	W =  -168.557 deg,	P =    -0.849 deg,	R =  -103.190 deg
};
P[1772]{
   GP1:
	UF : 7, UT : 3,	CONFIG : 'F U T, 0, 0, 0',
	X =  -284.464  mm,	Y =   167.284  mm,	Z =     0.271  mm,
	W =  -168.319 deg,	P =    -1.416 deg,	R =  -105.411 deg
};
P[1773]{
   GP1:
	UF : 7, UT : 3,	CONFIG : 'F U T, 0, 0, 0',
	X =  -279.044  mm,	Y =   176.157  mm,	Z =     0.000  mm,
	W =  -167.988 deg,	P =    -1.117 deg,	R =  -107.842 deg
};
P[1774]{
   GP1:
	UF : 7, UT : 3,	CONFIG : 'F U T, 0, 0, 0',
	X =  -279.044  mm,	Y =   176.157  mm,	Z =     0.000  mm,
	W =  -167.988 deg,	P =    -1.117 deg,	R =  -107.842 deg
};
P[1775]{
   GP1:
	UF : 7, UT : 3,	CONFIG : 'F U T, 0, 0, 0',
	X =  -279.044  mm,	Y =   176.157  mm,	Z =     0.000  mm,
	W =  -167.988 deg,	P =    -1.117 deg,	R =  -107.842 deg
};
P[1776]{
   GP1:
	UF : 7, UT : 3,	CONFIG : 'F U T, 0, 0, 0',
	X =  -279.044  mm,	Y =   176.157  mm,	Z =     0.000  mm,
	W =  -167.988 deg,	P =    -1.117 deg,	R =  -107.842 deg
};
P[1777]{
   GP1:
	UF : 7, UT : 3,	CONFIG : 'F U T, 0, 0, 0',
	X =  -233.834  mm,	Y =   232.850  mm,	Z =     0.000  mm,
	W =  -167.362 deg,	P =     0.113 deg,	R =  -119.512 deg
};
P[1778]{
   GP1:
	UF : 7, UT : 3,	CONFIG : 'F U T, 0, 0, 0',
	X =  -233.834  mm,	Y =   232.850  mm,	Z =     0.000  mm,
	W =  -167.362 deg,	P =     0.113 deg,	R =  -119.512 deg
};
P[1779]{
   GP1:
	UF : 7, UT : 3,	CONFIG : 'F U T, 0, 0, 0',
	X =  -233.834  mm,	Y =   232.850  mm,	Z =     0.000  mm,
	W =  -167.362 deg,	P =     0.113 deg,	R =  -119.512 deg
};
P[1780]{
   GP1:
	UF : 7, UT : 3,	CONFIG : 'F U T, 0, 0, 0',
	X =  -233.834  mm,	Y =   232.850  mm,	Z =     0.000  mm,
	W =  -167.362 deg,	P =     0.113 deg,	R =  -119.512 deg
};
P[1781]{
   GP1:
	UF : 7, UT : 3,	CONFIG : 'F U T, 0, 0, 0',
	X =  -223.959  mm,	Y =   242.372  mm,	Z =     0.017  mm,
	W =  -167.363 deg,	P =     0.051 deg,	R =  -122.203 deg
};
P[1782]{
   GP1:
	UF : 7, UT : 3,	CONFIG : 'F U T, 0, 0, 0',
	X =  -213.205  mm,	Y =   251.879  mm,	Z =     0.019  mm,
	W =  -167.357 deg,	P =    -0.013 deg,	R =  -124.752 deg
};
P[1783]{
   GP1:
	UF : 7, UT : 3,	CONFIG : 'F U T, 0, 0, 0',
	X =  -201.087  mm,	Y =   261.652  mm,	Z =     0.013  mm,
	W =  -167.362 deg,	P =    -0.013 deg,	R =  -127.460 deg
};
P[1784]{
   GP1:
	UF : 7, UT : 3,	CONFIG : 'F U T, 0, 0, 0',
	X =  -188.194  mm,	Y =   271.072  mm,	Z =     0.006  mm,
	W =  -167.366 deg,	P =    -0.013 deg,	R =  -130.104 deg
};
P[1785]{
   GP1:
	UF : 7, UT : 3,	CONFIG : 'F U T, 0, 0, 0',
	X =  -174.980  mm,	Y =   279.789  mm,	Z =     0.000  mm,
	W =  -167.371 deg,	P =    -0.013 deg,	R =  -132.787 deg
};
P[1786]{
   GP1:
	UF : 7, UT : 3,	CONFIG : 'F U T, 0, 0, 0',
	X =  -174.980  mm,	Y =   279.789  mm,	Z =     0.000  mm,
	W =  -167.371 deg,	P =    -0.013 deg,	R =  -132.787 deg
};
P[1787]{
   GP1:
	UF : 7, UT : 3,	CONFIG : 'F U T, 0, 0, 0',
	X =  -174.980  mm,	Y =   279.789  mm,	Z =     0.000  mm,
	W =  -167.371 deg,	P =    -0.013 deg,	R =  -132.787 deg
};
P[1788]{
   GP1:
	UF : 7, UT : 3,	CONFIG : 'F U T, 0, 0, 0',
	X =  -174.980  mm,	Y =   279.789  mm,	Z =     0.000  mm,
	W =  -167.371 deg,	P =    -0.013 deg,	R =  -132.787 deg
};
P[1789]{
   GP1:
	UF : 7, UT : 3,	CONFIG : 'F U T, 0, 0, 0',
	X =  -109.648  mm,	Y =   311.249  mm,	Z =     0.000  mm,
	W =  -167.363 deg,	P =     0.003 deg,	R =  -145.199 deg
};
P[1790]{
   GP1:
	UF : 7, UT : 3,	CONFIG : 'F U T, 0, 0, 0',
	X =  -109.648  mm,	Y =   311.249  mm,	Z =     0.000  mm,
	W =  -167.363 deg,	P =     0.003 deg,	R =  -145.199 deg
};
P[1791]{
   GP1:
	UF : 7, UT : 3,	CONFIG : 'F U T, 0, 0, 0',
	X =  -109.648  mm,	Y =   311.249  mm,	Z =     0.000  mm,
	W =  -167.363 deg,	P =     0.003 deg,	R =  -145.199 deg
};
P[1792]{
   GP1:
	UF : 7, UT : 3,	CONFIG : 'F U T, 0, 0, 0',
	X =  -109.648  mm,	Y =   311.249  mm,	Z =     0.000  mm,
	W =  -167.363 deg,	P =     0.003 deg,	R =  -145.199 deg
};
P[1793]{
   GP1:
	UF : 7, UT : 3,	CONFIG : 'F U T, 0, 0, 0',
	X =   -92.942  mm,	Y =   316.644  mm,	Z =     0.000  mm,
	W =  -167.364 deg,	P =     0.002 deg,	R =  -148.612 deg
};
P[1794]{
   GP1:
	UF : 7, UT : 3,	CONFIG : 'F U T, 0, 0, 0',
	X =   -74.994  mm,	Y =   321.366  mm,	Z =     0.000  mm,
	W =  -167.364 deg,	P =     0.001 deg,	R =  -151.812 deg
};
P[1795]{
   GP1:
	UF : 7, UT : 3,	CONFIG : 'F U T, 0, 0, 0',
	X =   -56.916  mm,	Y =   325.063  mm,	Z =     0.000  mm,
	W =  -167.364 deg,	P =     0.001 deg,	R =  -155.040 deg
};
P[1796]{
   GP1:
	UF : 7, UT : 3,	CONFIG : 'F U T, 0, 0, 0',
	X =   -36.254  mm,	Y =   328.016  mm,	Z =     0.000  mm,
	W =  -167.364 deg,	P =     0.000 deg,	R =  -158.080 deg
};
P[1797]{
   GP1:
	UF : 7, UT : 3,	CONFIG : 'F U T, 0, 0, 0',
	X =   -36.254  mm,	Y =   328.016  mm,	Z =     0.000  mm,
	W =  -167.364 deg,	P =     0.000 deg,	R =  -158.080 deg
};
P[1798]{
   GP1:
	UF : 7, UT : 3,	CONFIG : 'F U T, 0, 0, 0',
	X =   -36.254  mm,	Y =   328.016  mm,	Z =     0.000  mm,
	W =  -167.364 deg,	P =     0.000 deg,	R =  -158.080 deg
};
P[1799]{
   GP1:
	UF : 7, UT : 3,	CONFIG : 'F U T, 0, 0, 0',
	X =   -36.254  mm,	Y =   328.016  mm,	Z =     0.000  mm,
	W =  -167.364 deg,	P =     0.000 deg,	R =  -158.080 deg
};
P[1800]{
   GP1:
	UF : 7, UT : 3,	CONFIG : 'F U T, 0, 0, 0',
	X =    36.254  mm,	Y =   328.016  mm,	Z =     0.000  mm,
	W =  -167.363 deg,	P =     0.000 deg,	R =  -171.814 deg
};
P[1801]{
   GP1:
	UF : 7, UT : 3,	CONFIG : 'F U T, 0, 0, 0',
	X =    36.254  mm,	Y =   328.016  mm,	Z =     0.000  mm,
	W =  -167.363 deg,	P =     0.000 deg,	R =  -171.814 deg
};
P[1802]{
   GP1:
	UF : 7, UT : 3,	CONFIG : 'F U T, 0, 0, 0',
	X =    36.254  mm,	Y =   328.016  mm,	Z =     0.000  mm,
	W =  -167.363 deg,	P =     0.000 deg,	R =  -171.814 deg
};
P[1803]{
   GP1:
	UF : 7, UT : 3,	CONFIG : 'F U T, 0, 0, 0',
	X =    36.254  mm,	Y =   328.016  mm,	Z =     0.000  mm,
	W =  -167.363 deg,	P =     0.000 deg,	R =  -171.814 deg
};
P[1804]{
   GP1:
	UF : 7, UT : 3,	CONFIG : 'F U T, 0, 0, 0',
	X =    56.849  mm,	Y =   325.071  mm,	Z =     0.000  mm,
	W =  -167.364 deg,	P =     0.000 deg,	R =  -174.875 deg
};
P[1805]{
   GP1:
	UF : 7, UT : 3,	CONFIG : 'F U T, 0, 0, 0',
	X =    75.000  mm,	Y =   321.364  mm,	Z =     0.000  mm,
	W =  -167.364 deg,	P =     0.000 deg,	R =  -178.084 deg
};
P[1806]{
   GP1:
	UF : 7, UT : 3,	CONFIG : 'F U T, 0, 0, 0',
	X =    92.941  mm,	Y =   316.644  mm,	Z =     0.000  mm,
	W =  -167.364 deg,	P =     0.000 deg,	R =   178.713 deg
};
P[1807]{
   GP1:
	UF : 7, UT : 3,	CONFIG : 'F U T, 0, 0, 0',
	X =   109.648  mm,	Y =   311.249  mm,	Z =     0.000  mm,
	W =  -167.364 deg,	P =     0.000 deg,	R =   175.300 deg
};
P[1808]{
   GP1:
	UF : 7, UT : 3,	CONFIG : 'F U T, 0, 0, 0',
	X =   109.648  mm,	Y =   311.249  mm,	Z =     0.000  mm,
	W =  -167.364 deg,	P =     0.000 deg,	R =   175.300 deg
};
P[1809]{
   GP1:
	UF : 7, UT : 3,	CONFIG : 'F U T, 0, 0, 0',
	X =   109.648  mm,	Y =   311.249  mm,	Z =     0.000  mm,
	W =  -167.364 deg,	P =     0.000 deg,	R =   175.300 deg
};
P[1810]{
   GP1:
	UF : 7, UT : 3,	CONFIG : 'F U T, 0, 0, 0',
	X =   109.648  mm,	Y =   311.249  mm,	Z =     0.000  mm,
	W =  -167.364 deg,	P =     0.000 deg,	R =   175.300 deg
};
P[1811]{
   GP1:
	UF : 7, UT : 3,	CONFIG : 'F U T, 0, 0, 0',
	X =   174.980  mm,	Y =   279.789  mm,	Z =     0.000  mm,
	W =  -167.363 deg,	P =     0.001 deg,	R =   163.044 deg
};
P[1812]{
   GP1:
	UF : 7, UT : 3,	CONFIG : 'F U T, 0, 0, 0',
	X =   174.980  mm,	Y =   279.789  mm,	Z =     0.000  mm,
	W =  -167.363 deg,	P =     0.001 deg,	R =   163.044 deg
};
P[1813]{
   GP1:
	UF : 7, UT : 3,	CONFIG : 'F U T, 0, 0, 0',
	X =   174.980  mm,	Y =   279.789  mm,	Z =     0.000  mm,
	W =  -167.363 deg,	P =     0.001 deg,	R =   163.044 deg
};
P[1814]{
   GP1:
	UF : 7, UT : 3,	CONFIG : 'F U T, 0, 0, 0',
	X =   174.980  mm,	Y =   279.789  mm,	Z =     0.000  mm,
	W =  -167.363 deg,	P =     0.001 deg,	R =   163.044 deg
};
P[1815]{
   GP1:
	UF : 7, UT : 3,	CONFIG : 'F U T, 0, 0, 0',
	X =   190.679  mm,	Y =   269.339  mm,	Z =     0.000  mm,
	W =  -167.364 deg,	P =     0.001 deg,	R =   159.762 deg
};
P[1816]{
   GP1:
	UF : 7, UT : 3,	CONFIG : 'F U T, 0, 0, 0',
	X =   205.753  mm,	Y =   258.007  mm,	Z =     0.000  mm,
	W =  -167.364 deg,	P =     0.000 deg,	R =   156.479 deg
};
P[1817]{
   GP1:
	UF : 7, UT : 3,	CONFIG : 'F U T, 0, 0, 0',
	X =   220.154  mm,	Y =   245.831  mm,	Z =     0.000  mm,
	W =  -167.364 deg,	P =    -0.001 deg,	R =   153.196 deg
};
P[1818]{
   GP1:
	UF : 7, UT : 3,	CONFIG : 'F U T, 0, 0, 0',
	X =   233.834  mm,	Y =   232.850  mm,	Z =     0.000  mm,
	W =  -167.365 deg,	P =    -0.002 deg,	R =   149.914 deg
};
P[1819]{
   GP1:
	UF : 7, UT : 3,	CONFIG : 'F U T, 0, 0, 0',
	X =   233.834  mm,	Y =   232.850  mm,	Z =     0.000  mm,
	W =  -167.365 deg,	P =    -0.002 deg,	R =   149.914 deg
};
P[1820]{
   GP1:
	UF : 7, UT : 3,	CONFIG : 'F U T, 0, 0, 0',
	X =   233.834  mm,	Y =   232.850  mm,	Z =     0.000  mm,
	W =  -167.365 deg,	P =    -0.002 deg,	R =   149.914 deg
};
P[1821]{
   GP1:
	UF : 7, UT : 3,	CONFIG : 'F U T, 0, 0, 0',
	X =   233.834  mm,	Y =   232.850  mm,	Z =     0.000  mm,
	W =  -167.365 deg,	P =    -0.002 deg,	R =   149.914 deg
};
P[1822]{
   GP1:
	UF : 7, UT : 3,	CONFIG : 'F U T, 0, 0, 0',
	X =   279.044  mm,	Y =   176.157  mm,	Z =     0.000  mm,
	W =  -167.363 deg,	P =     0.002 deg,	R =   137.857 deg
};
P[1823]{
   GP1:
	UF : 7, UT : 3,	CONFIG : 'F U T, 0, 0, 0',
	X =   279.044  mm,	Y =   176.157  mm,	Z =     0.000  mm,
	W =  -167.363 deg,	P =     0.002 deg,	R =   137.857 deg
};
P[1824]{
   GP1:
	UF : 7, UT : 3,	CONFIG : 'F U T, 0, 0, 0',
	X =   279.044  mm,	Y =   176.157  mm,	Z =     0.000  mm,
	W =  -167.363 deg,	P =     0.002 deg,	R =   137.857 deg
};
P[1825]{
   GP1:
	UF : 7, UT : 3,	CONFIG : 'F U T, 0, 0, 0',
	X =   279.044  mm,	Y =   176.157  mm,	Z =     0.000  mm,
	W =  -167.363 deg,	P =     0.002 deg,	R =   137.857 deg
};
P[1826]{
   GP1:
	UF : 7, UT : 3,	CONFIG : 'F U T, 0, 0, 0',
	X =   287.893  mm,	Y =   161.305  mm,	Z =     0.000  mm,
	W =  -167.364 deg,	P =     0.001 deg,	R =   134.332 deg
};
P[1827]{
   GP1:
	UF : 7, UT : 3,	CONFIG : 'F U T, 0, 0, 0',
	X =   296.479  mm,	Y =   144.911  mm,	Z =     0.000  mm,
	W =  -167.364 deg,	P =     0.000 deg,	R =   131.099 deg
};
P[1828]{
   GP1:
	UF : 7, UT : 3,	CONFIG : 'F U T, 0, 0, 0',
	X =   304.165  mm,	Y =   128.012  mm,	Z =     0.000  mm,
	W =  -167.364 deg,	P =    -0.001 deg,	R =   127.883 deg
};
P[1829]{
   GP1:
	UF : 7, UT : 3,	CONFIG : 'F U T, 0, 0, 0',
	X =   311.718  mm,	Y =   108.335  mm,	Z =     0.000  mm,
	W =  -167.365 deg,	P =    -0.002 deg,	R =   124.706 deg
};
P[1830]{
   GP1:
	UF : 7, UT : 3,	CONFIG : 'F U T, 0, 0, 0',
	X =   311.718  mm,	Y =   108.335  mm,	Z =     0.000  mm,
	W =  -167.365 deg,	P =    -0.002 deg,	R =   124.706 deg
};
P[1831]{
   GP1:
	UF : 7, UT : 3,	CONFIG : 'F U T, 0, 0, 0',
	X =   311.718  mm,	Y =   108.335  mm,	Z =     0.000  mm,
	W =  -167.365 deg,	P =    -0.002 deg,	R =   124.706 deg
};
P[1832]{
   GP1:
	UF : 7, UT : 3,	CONFIG : 'F U T, 0, 0, 0',
	X =   311.718  mm,	Y =   108.335  mm,	Z =     0.000  mm,
	W =  -167.365 deg,	P =    -0.002 deg,	R =   124.706 deg
};
P[1833]{
   GP1:
	UF : 7, UT : 3,	CONFIG : 'F U T, 0, 0, 0',
	X =   327.850  mm,	Y =    37.642  mm,	Z =     0.000  mm,
	W =  -167.363 deg,	P =     0.001 deg,	R =   111.494 deg
};
P[1834]{
   GP1:
	UF : 7, UT : 3,	CONFIG : 'F U T, 0, 0, 0',
	X =   327.850  mm,	Y =    37.642  mm,	Z =     0.000  mm,
	W =  -167.363 deg,	P =     0.001 deg,	R =   111.494 deg
};
P[1835]{
   GP1:
	UF : 7, UT : 3,	CONFIG : 'F U T, 0, 0, 0',
	X =   327.850  mm,	Y =    37.642  mm,	Z =     0.000  mm,
	W =  -167.363 deg,	P =     0.001 deg,	R =   111.494 deg
};
P[1836]{
   GP1:
	UF : 7, UT : 3,	CONFIG : 'F U T, 0, 0, 0',
	X =   327.850  mm,	Y =    37.642  mm,	Z =     0.000  mm,
	W =  -167.363 deg,	P =     0.001 deg,	R =   111.494 deg
};
P[1837]{
   GP1:
	UF : 7, UT : 3,	CONFIG : 'F U T, 0, 0, 0',
	X =   329.392  mm,	Y =    20.047  mm,	Z =     0.000  mm,
	W =  -167.364 deg,	P =     0.000 deg,	R =   108.496 deg
};
P[1838]{
   GP1:
	UF : 7, UT : 3,	CONFIG : 'F U T, 0, 0, 0',
	X =   330.015  mm,	Y =     0.000  mm,	Z =     0.000  mm,
	W =  -167.364 deg,	P =    -0.001 deg,	R =   105.709 deg
};
P[1839]{
   GP1:
	UF : 7, UT : 3,	CONFIG : 'F U T, 0, 0, 0',
	X =   330.015  mm,	Y =     0.000  mm,	Z =     0.000  mm,
	W =  -167.364 deg,	P =    -0.001 deg,	R =   105.709 deg
};
P[1840]{
   GP1:
	UF : 7, UT : 3,	CONFIG : 'F U T, 0, 0, 0',
	X =   330.015  mm,	Y =     0.000  mm,	Z =     0.000  mm,
	W =  -167.364 deg,	P =    -0.001 deg,	R =   105.709 deg
};
P[1841]{
   GP1:
	UF : 7, UT : 3,	CONFIG : 'F U T, 0, 0, 0',
	X =   330.015  mm,	Y =     0.000  mm,	Z =     0.000  mm,
	W =  -167.364 deg,	P =    -0.001 deg,	R =   105.709 deg
};
P[1842]{
   GP1:
	UF : 7, UT : 3,	CONFIG : 'F U T, 0, 0, 0',
	X =   326.881  mm,	Y =     0.000  mm,	Z =     0.000  mm,
	W =  -167.364 deg,	P =    -0.001 deg,	R =   105.719 deg
};
P[1843]{
   GP1:
	UF : 7, UT : 3,	CONFIG : 'F U T, 0, 0, 0',
	X =   326.881  mm,	Y =     0.000  mm,	Z =     0.000  mm,
	W =  -167.364 deg,	P =    -0.001 deg,	R =   105.719 deg
};
P[1844]{
   GP1:
	UF : 7, UT : 3,	CONFIG : 'F U T, 0, 0, 0',
	X =   326.881  mm,	Y =     0.000  mm,	Z =     0.000  mm,
	W =  -167.364 deg,	P =    -0.001 deg,	R =   105.719 deg
};
P[1845]{
   GP1:
	UF : 7, UT : 3,	CONFIG : 'F U T, 0, 0, 0',
	X =   326.881  mm,	Y =     0.000  mm,	Z =     0.000  mm,
	W =  -167.364 deg,	P =    -0.001 deg,	R =   105.719 deg
};
P[1846]{
   GP1:
	UF : 7, UT : 3,	CONFIG : 'F U T, 0, 0, 0',
	X =   326.322  mm,	Y =    18.789  mm,	Z =     0.000  mm,
	W =  -167.364 deg,	P =     0.000 deg,	R =   108.339 deg
};
P[1847]{
   GP1:
	UF : 7, UT : 3,	CONFIG : 'F U T, 0, 0, 0',
	X =   324.819  mm,	Y =    36.609  mm,	Z =     0.000  mm,
	W =  -167.363 deg,	P =     0.001 deg,	R =   111.080 deg
};
P[1848]{
   GP1:
	UF : 7, UT : 3,	CONFIG : 'F U T, 0, 0, 0',
	X =   324.819  mm,	Y =    36.609  mm,	Z =     0.000  mm,
	W =  -167.363 deg,	P =     0.001 deg,	R =   111.080 deg
};
P[1849]{
   GP1:
	UF : 7, UT : 3,	CONFIG : 'F U T, 0, 0, 0',
	X =   324.819  mm,	Y =    36.609  mm,	Z =     0.000  mm,
	W =  -167.363 deg,	P =     0.001 deg,	R =   111.080 deg
};
P[1850]{
   GP1:
	UF : 7, UT : 3,	CONFIG : 'F U T, 0, 0, 0',
	X =   324.819  mm,	Y =    36.609  mm,	Z =     0.000  mm,
	W =  -167.363 deg,	P =     0.001 deg,	R =   111.080 deg
};
P[1851]{
   GP1:
	UF : 7, UT : 3,	CONFIG : 'F U T, 0, 0, 0',
	X =   308.528  mm,	Y =   107.949  mm,	Z =     0.000  mm,
	W =  -167.365 deg,	P =    -0.002 deg,	R =   124.620 deg
};
P[1852]{
   GP1:
	UF : 7, UT : 3,	CONFIG : 'F U T, 0, 0, 0',
	X =   308.528  mm,	Y =   107.949  mm,	Z =     0.000  mm,
	W =  -167.365 deg,	P =    -0.002 deg,	R =   124.620 deg
};
P[1853]{
   GP1:
	UF : 7, UT : 3,	CONFIG : 'F U T, 0, 0, 0',
	X =   308.528  mm,	Y =   107.949  mm,	Z =     0.000  mm,
	W =  -167.365 deg,	P =    -0.002 deg,	R =   124.620 deg
};
P[1854]{
   GP1:
	UF : 7, UT : 3,	CONFIG : 'F U T, 0, 0, 0',
	X =   308.528  mm,	Y =   107.949  mm,	Z =     0.000  mm,
	W =  -167.365 deg,	P =    -0.002 deg,	R =   124.620 deg
};
P[1855]{
   GP1:
	UF : 7, UT : 3,	CONFIG : 'F U T, 0, 0, 0',
	X =   301.533  mm,	Y =   126.177  mm,	Z =     0.001  mm,
	W =  -167.364 deg,	P =    -0.001 deg,	R =   127.743 deg
};
P[1856]{
   GP1:
	UF : 7, UT : 3,	CONFIG : 'F U T, 0, 0, 0',
	X =   293.998  mm,	Y =   142.847  mm,	Z =     0.000  mm,
	W =  -167.364 deg,	P =     0.000 deg,	R =   130.977 deg
};
P[1857]{
   GP1:
	UF : 7, UT : 3,	CONFIG : 'F U T, 0, 0, 0',
	X =   285.500  mm,	Y =   159.164  mm,	Z =     0.000  mm,
	W =  -167.364 deg,	P =     0.001 deg,	R =   134.192 deg
};
P[1858]{
   GP1:
	UF : 7, UT : 3,	CONFIG : 'F U T, 0, 0, 0',
	X =   276.758  mm,	Y =   173.908  mm,	Z =     0.000  mm,
	W =  -167.363 deg,	P =     0.002 deg,	R =   137.706 deg
};
P[1859]{
   GP1:
	UF : 7, UT : 3,	CONFIG : 'F U T, 0, 0, 0',
	X =   276.758  mm,	Y =   173.908  mm,	Z =     0.000  mm,
	W =  -167.363 deg,	P =     0.002 deg,	R =   137.706 deg
};
P[1860]{
   GP1:
	UF : 7, UT : 3,	CONFIG : 'F U T, 0, 0, 0',
	X =   276.758  mm,	Y =   173.908  mm,	Z =     0.000  mm,
	W =  -167.363 deg,	P =     0.002 deg,	R =   137.706 deg
};
P[1861]{
   GP1:
	UF : 7, UT : 3,	CONFIG : 'F U T, 0, 0, 0',
	X =   276.758  mm,	Y =   173.908  mm,	Z =     0.000  mm,
	W =  -167.363 deg,	P =     0.002 deg,	R =   137.706 deg
};
P[1862]{
   GP1:
	UF : 7, UT : 3,	CONFIG : 'F U T, 0, 0, 0',
	X =   231.131  mm,	Y =   231.120  mm,	Z =     0.000  mm,
	W =  -167.364 deg,	P =    -0.002 deg,	R =   149.652 deg
};
P[1863]{
   GP1:
	UF : 7, UT : 3,	CONFIG : 'F U T, 0, 0, 0',
	X =   231.131  mm,	Y =   231.120  mm,	Z =     0.000  mm,
	W =  -167.364 deg,	P =    -0.002 deg,	R =   149.652 deg
};
P[1864]{
   GP1:
	UF : 7, UT : 3,	CONFIG : 'F U T, 0, 0, 0',
	X =   231.131  mm,	Y =   231.120  mm,	Z =     0.000  mm,
	W =  -167.364 deg,	P =    -0.002 deg,	R =   149.652 deg
};
P[1865]{
   GP1:
	UF : 7, UT : 3,	CONFIG : 'F U T, 0, 0, 0',
	X =   231.131  mm,	Y =   231.120  mm,	Z =     0.000  mm,
	W =  -167.364 deg,	P =    -0.002 deg,	R =   149.652 deg
};
P[1866]{
   GP1:
	UF : 7, UT : 3,	CONFIG : 'F U T, 0, 0, 0',
	X =   218.314  mm,	Y =   243.276  mm,	Z =     0.001  mm,
	W =  -167.364 deg,	P =    -0.001 deg,	R =   153.151 deg
};
P[1867]{
   GP1:
	UF : 7, UT : 3,	CONFIG : 'F U T, 0, 0, 0',
	X =   203.983  mm,	Y =   255.400  mm,	Z =     0.001  mm,
	W =  -167.364 deg,	P =     0.000 deg,	R =   156.409 deg
};
P[1868]{
   GP1:
	UF : 7, UT : 3,	CONFIG : 'F U T, 0, 0, 0',
	X =   189.201  mm,	Y =   266.552  mm,	Z =     0.001  mm,
	W =  -167.364 deg,	P =     0.001 deg,	R =   159.717 deg
};
P[1869]{
   GP1:
	UF : 7, UT : 3,	CONFIG : 'F U T, 0, 0, 0',
	X =   173.895  mm,	Y =   276.767  mm,	Z =     0.000  mm,
	W =  -167.363 deg,	P =     0.002 deg,	R =   163.034 deg
};
P[1870]{
   GP1:
	UF : 7, UT : 3,	CONFIG : 'F U T, 0, 0, 0',
	X =   173.895  mm,	Y =   276.767  mm,	Z =     0.000  mm,
	W =  -167.363 deg,	P =     0.002 deg,	R =   163.034 deg
};
P[1871]{
   GP1:
	UF : 7, UT : 3,	CONFIG : 'F U T, 0, 0, 0',
	X =   173.895  mm,	Y =   276.767  mm,	Z =     0.000  mm,
	W =  -167.363 deg,	P =     0.002 deg,	R =   163.034 deg
};
P[1872]{
   GP1:
	UF : 7, UT : 3,	CONFIG : 'F U T, 0, 0, 0',
	X =   173.895  mm,	Y =   276.767  mm,	Z =     0.000  mm,
	W =  -167.363 deg,	P =     0.002 deg,	R =   163.034 deg
};
P[1873]{
   GP1:
	UF : 7, UT : 3,	CONFIG : 'F U T, 0, 0, 0',
	X =   107.966  mm,	Y =   308.522  mm,	Z =     0.000  mm,
	W =  -167.364 deg,	P =     0.000 deg,	R =   175.671 deg
};
P[1874]{
   GP1:
	UF : 7, UT : 3,	CONFIG : 'F U T, 0, 0, 0',
	X =   107.966  mm,	Y =   308.522  mm,	Z =     0.000  mm,
	W =  -167.364 deg,	P =     0.000 deg,	R =   175.671 deg
};
P[1875]{
   GP1:
	UF : 7, UT : 3,	CONFIG : 'F U T, 0, 0, 0',
	X =   107.966  mm,	Y =   308.522  mm,	Z =     0.000  mm,
	W =  -167.364 deg,	P =     0.000 deg,	R =   175.671 deg
};
P[1876]{
   GP1:
	UF : 7, UT : 3,	CONFIG : 'F U T, 0, 0, 0',
	X =   107.966  mm,	Y =   308.522  mm,	Z =     0.000  mm,
	W =  -167.364 deg,	P =     0.000 deg,	R =   175.671 deg
};
P[1877]{
   GP1:
	UF : 7, UT : 3,	CONFIG : 'F U T, 0, 0, 0',
	X =    91.343  mm,	Y =   313.844  mm,	Z =     0.000  mm,
	W =  -167.364 deg,	P =     0.000 deg,	R =   178.849 deg
};
P[1878]{
   GP1:
	UF : 7, UT : 3,	CONFIG : 'F U T, 0, 0, 0',
	X =    74.067  mm,	Y =   318.365  mm,	Z =     0.000  mm,
	W =  -167.364 deg,	P =     0.000 deg,	R =  -178.042 deg
};
P[1879]{
   GP1:
	UF : 7, UT : 3,	CONFIG : 'F U T, 0, 0, 0',
	X =    56.672  mm,	Y =   321.921  mm,	Z =     0.000  mm,
	W =  -167.364 deg,	P =     0.000 deg,	R =  -174.914 deg
};
P[1880]{
   GP1:
	UF : 7, UT : 3,	CONFIG : 'F U T, 0, 0, 0',
	X =    36.588  mm,	Y =   324.822  mm,	Z =     0.000  mm,
	W =  -167.363 deg,	P =     0.000 deg,	R =  -171.929 deg
};
P[1881]{
   GP1:
	UF : 7, UT : 3,	CONFIG : 'F U T, 0, 0, 0',
	X =    36.588  mm,	Y =   324.822  mm,	Z =     0.000  mm,
	W =  -167.363 deg,	P =     0.000 deg,	R =  -171.929 deg
};
P[1882]{
   GP1:
	UF : 7, UT : 3,	CONFIG : 'F U T, 0, 0, 0',
	X =    36.588  mm,	Y =   324.822  mm,	Z =     0.000  mm,
	W =  -167.363 deg,	P =     0.000 deg,	R =  -171.929 deg
};
P[1883]{
   GP1:
	UF : 7, UT : 3,	CONFIG : 'F U T, 0, 0, 0',
	X =    36.588  mm,	Y =   324.822  mm,	Z =     0.000  mm,
	W =  -167.363 deg,	P =     0.000 deg,	R =  -171.929 deg
};
P[1884]{
   GP1:
	UF : 7, UT : 3,	CONFIG : 'F U T, 0, 0, 0',
	X =   -36.588  mm,	Y =   324.822  mm,	Z =     0.000  mm,
	W =  -167.364 deg,	P =    -0.001 deg,	R =  -157.966 deg
};
P[1885]{
   GP1:
	UF : 7, UT : 3,	CONFIG : 'F U T, 0, 0, 0',
	X =   -36.588  mm,	Y =   324.822  mm,	Z =     0.000  mm,
	W =  -167.364 deg,	P =    -0.001 deg,	R =  -157.966 deg
};
P[1886]{
   GP1:
	UF : 7, UT : 3,	CONFIG : 'F U T, 0, 0, 0',
	X =   -36.588  mm,	Y =   324.822  mm,	Z =     0.000  mm,
	W =  -167.364 deg,	P =    -0.001 deg,	R =  -157.966 deg
};
P[1887]{
   GP1:
	UF : 7, UT : 3,	CONFIG : 'F U T, 0, 0, 0',
	X =   -36.588  mm,	Y =   324.822  mm,	Z =     0.000  mm,
	W =  -167.364 deg,	P =    -0.001 deg,	R =  -157.966 deg
};
P[1888]{
   GP1:
	UF : 7, UT : 3,	CONFIG : 'F U T, 0, 0, 0',
	X =   -56.735  mm,	Y =   321.912  mm,	Z =     0.000  mm,
	W =  -167.364 deg,	P =     0.001 deg,	R =  -154.974 deg
};
P[1889]{
   GP1:
	UF : 7, UT : 3,	CONFIG : 'F U T, 0, 0, 0',
	X =   -74.092  mm,	Y =   318.359  mm,	Z =     0.000  mm,
	W =  -167.364 deg,	P =     0.001 deg,	R =  -151.851 deg
};
P[1890]{
   GP1:
	UF : 7, UT : 3,	CONFIG : 'F U T, 0, 0, 0',
	X =   -91.376  mm,	Y =   313.835  mm,	Z =     0.001  mm,
	W =  -167.363 deg,	P =     0.002 deg,	R =  -148.753 deg
};
P[1891]{
   GP1:
	UF : 7, UT : 3,	CONFIG : 'F U T, 0, 0, 0',
	X =  -107.966  mm,	Y =   308.522  mm,	Z =     0.000  mm,
	W =  -167.363 deg,	P =     0.003 deg,	R =  -145.585 deg
};
P[1892]{
   GP1:
	UF : 7, UT : 3,	CONFIG : 'F U T, 0, 0, 0',
	X =  -107.966  mm,	Y =   308.522  mm,	Z =     0.000  mm,
	W =  -167.363 deg,	P =     0.003 deg,	R =  -145.585 deg
};
P[1893]{
   GP1:
	UF : 7, UT : 3,	CONFIG : 'F U T, 0, 0, 0',
	X =  -107.966  mm,	Y =   308.522  mm,	Z =     0.000  mm,
	W =  -167.363 deg,	P =     0.003 deg,	R =  -145.585 deg
};
P[1894]{
   GP1:
	UF : 7, UT : 3,	CONFIG : 'F U T, 0, 0, 0',
	X =  -107.966  mm,	Y =   308.522  mm,	Z =     0.000  mm,
	W =  -167.363 deg,	P =     0.003 deg,	R =  -145.585 deg
};
P[1895]{
   GP1:
	UF : 7, UT : 3,	CONFIG : 'F U T, 0, 0, 0',
	X =  -173.895  mm,	Y =   276.767  mm,	Z =     0.000  mm,
	W =  -167.370 deg,	P =    -0.015 deg,	R =  -132.924 deg
};
P[1896]{
   GP1:
	UF : 7, UT : 3,	CONFIG : 'F U T, 0, 0, 0',
	X =  -173.895  mm,	Y =   276.767  mm,	Z =     0.000  mm,
	W =  -167.370 deg,	P =    -0.015 deg,	R =  -132.924 deg
};
P[1897]{
   GP1:
	UF : 7, UT : 3,	CONFIG : 'F U T, 0, 0, 0',
	X =  -173.895  mm,	Y =   276.767  mm,	Z =     0.000  mm,
	W =  -167.370 deg,	P =    -0.015 deg,	R =  -132.924 deg
};
P[1898]{
   GP1:
	UF : 7, UT : 3,	CONFIG : 'F U T, 0, 0, 0',
	X =  -173.895  mm,	Y =   276.767  mm,	Z =     0.000  mm,
	W =  -167.370 deg,	P =    -0.015 deg,	R =  -132.924 deg
};
P[1899]{
   GP1:
	UF : 7, UT : 3,	CONFIG : 'F U T, 0, 0, 0',
	X =  -186.182  mm,	Y =   268.655  mm,	Z =     0.005  mm,
	W =  -167.365 deg,	P =    -0.015 deg,	R =  -130.212 deg
};
P[1900]{
   GP1:
	UF : 7, UT : 3,	CONFIG : 'F U T, 0, 0, 0',
	X =  -198.498  mm,	Y =   259.687  mm,	Z =     0.013  mm,
	W =  -167.359 deg,	P =    -0.015 deg,	R =  -127.581 deg
};
P[1901]{
   GP1:
	UF : 7, UT : 3,	CONFIG : 'F U T, 0, 0, 0',
	X =  -210.302  mm,	Y =   250.226  mm,	Z =     0.019  mm,
	W =  -167.354 deg,	P =    -0.016 deg,	R =  -124.938 deg
};
P[1902]{
   GP1:
	UF : 7, UT : 3,	CONFIG : 'F U T, 0, 0, 0',
	X =  -221.274  mm,	Y =   240.579  mm,	Z =     0.017  mm,
	W =  -167.356 deg,	P =     0.051 deg,	R =  -122.320 deg
};
P[1903]{
   GP1:
	UF : 7, UT : 3,	CONFIG : 'F U T, 0, 0, 0',
	X =  -231.131  mm,	Y =   231.120  mm,	Z =     0.000  mm,
	W =  -167.352 deg,	P =     0.114 deg,	R =  -119.469 deg
};
P[1904]{
   GP1:
	UF : 7, UT : 3,	CONFIG : 'F U T, 0, 0, 0',
	X =  -231.131  mm,	Y =   231.120  mm,	Z =     0.000  mm,
	W =  -167.352 deg,	P =     0.114 deg,	R =  -119.469 deg
};
P[1905]{
   GP1:
	UF : 7, UT : 3,	CONFIG : 'F U T, 0, 0, 0',
	X =  -231.131  mm,	Y =   231.120  mm,	Z =     0.000  mm,
	W =  -167.352 deg,	P =     0.114 deg,	R =  -119.469 deg
};
P[1906]{
   GP1:
	UF : 7, UT : 3,	CONFIG : 'F U T, 0, 0, 0',
	X =  -231.131  mm,	Y =   231.120  mm,	Z =     0.000  mm,
	W =  -167.352 deg,	P =     0.114 deg,	R =  -119.469 deg
};
P[1907]{
   GP1:
	UF : 7, UT : 3,	CONFIG : 'F U T, 0, 0, 0',
	X =  -276.758  mm,	Y =   173.908  mm,	Z =     0.000  mm,
	W =  -167.890 deg,	P =    -1.161 deg,	R =  -107.650 deg
};
P[1908]{
   GP1:
	UF : 7, UT : 3,	CONFIG : 'F U T, 0, 0, 0',
	X =  -276.758  mm,	Y =   173.908  mm,	Z =     0.000  mm,
	W =  -167.890 deg,	P =    -1.161 deg,	R =  -107.650 deg
};
P[1909]{
   GP1:
	UF : 7, UT : 3,	CONFIG : 'F U T, 0, 0, 0',
	X =  -276.758  mm,	Y =   173.908  mm,	Z =     0.000  mm,
	W =  -167.890 deg,	P =    -1.161 deg,	R =  -107.650 deg
};
P[1910]{
   GP1:
	UF : 7, UT : 3,	CONFIG : 'F U T, 0, 0, 0',
	X =  -276.758  mm,	Y =   173.908  mm,	Z =     0.000  mm,
	W =  -167.890 deg,	P =    -1.161 deg,	R =  -107.650 deg
};
P[1911]{
   GP1:
	UF : 7, UT : 3,	CONFIG : 'F U T, 0, 0, 0',
	X =  -282.022  mm,	Y =   165.259  mm,	Z =     0.257  mm,
	W =  -168.223 deg,	P =    -1.349 deg,	R =  -105.300 deg
};
P[1912]{
   GP1:
	UF : 7, UT : 3,	CONFIG : 'F U T, 0, 0, 0',
	X =  -288.425  mm,	Y =   153.813  mm,	Z =     0.563  mm,
	W =  -168.481 deg,	P =    -0.762 deg,	R =  -103.051 deg
};
P[1913]{
   GP1:
	UF : 7, UT : 3,	CONFIG : 'F U T, 0, 0, 0',
	X =  -296.971  mm,	Y =   136.562  mm,	Z =     0.670  mm,
	W =  -168.382 deg,	P =     0.631 deg,	R =   -99.690 deg
};
P[1914]{
   GP1:
	UF : 7, UT : 3,	CONFIG : 'F U T, 0, 0, 0',
	X =  -302.664  mm,	Y =   123.431  mm,	Z =     0.424  mm,
	W =  -167.898 deg,	P =     1.805 deg,	R =   -97.151 deg
};
P[1915]{
   GP1:
	UF : 7, UT : 3,	CONFIG : 'F U T, 0, 0, 0',
	X =  -305.358  mm,	Y =   116.596  mm,	Z =     0.206  mm,
	W =  -167.520 deg,	P =     1.756 deg,	R =   -95.843 deg
};
P[1916]{
   GP1:
	UF : 7, UT : 3,	CONFIG : 'F U T, 0, 0, 0',
	X =  -308.528  mm,	Y =   107.949  mm,	Z =     0.000  mm,
	W =  -167.297 deg,	P =     0.804 deg,	R =   -94.511 deg
};
P[1917]{
   GP1:
	UF : 7, UT : 3,	CONFIG : 'F U T, 0, 0, 0',
	X =  -308.528  mm,	Y =   107.949  mm,	Z =     0.000  mm,
	W =  -167.297 deg,	P =     0.804 deg,	R =   -94.511 deg
};
P[1918]{
   GP1:
	UF : 7, UT : 3,	CONFIG : 'F U T, 0, 0, 0',
	X =  -308.528  mm,	Y =   107.949  mm,	Z =     0.000  mm,
	W =  -167.297 deg,	P =     0.804 deg,	R =   -94.511 deg
};
P[1919]{
   GP1:
	UF : 7, UT : 3,	CONFIG : 'F U T, 0, 0, 0',
	X =  -308.528  mm,	Y =   107.949  mm,	Z =     0.000  mm,
	W =  -167.297 deg,	P =     0.804 deg,	R =   -94.511 deg
};
P[1920]{
   GP1:
	UF : 7, UT : 3,	CONFIG : 'F U T, 0, 1, 0',
	X =  -324.819  mm,	Y =    36.609  mm,	Z =     0.000  mm,
	W =  -167.369 deg,	P =    -0.011 deg,	R =   -80.976 deg
};
P[1921]{
   GP1:
	UF : 7, UT : 3,	CONFIG : 'F U T, 0, 1, 0',
	X =  -324.819  mm,	Y =    36.609  mm,	Z =     0.000  mm,
	W =  -167.369 deg,	P =    -0.011 deg,	R =   -80.976 deg
};
P[1922]{
   GP1:
	UF : 7, UT : 3,	CONFIG : 'F U T, 0, 1, 0',
	X =  -324.819  mm,	Y =    36.609  mm,	Z =     0.000  mm,
	W =  -167.369 deg,	P =    -0.011 deg,	R =   -80.976 deg
};
P[1923]{
   GP1:
	UF : 7, UT : 3,	CONFIG : 'F U T, 0, 1, 0',
	X =  -324.819  mm,	Y =    36.609  mm,	Z =     0.000  mm,
	W =  -167.369 deg,	P =    -0.011 deg,	R =   -80.976 deg
};
P[1924]{
   GP1:
	UF : 7, UT : 3,	CONFIG : 'F U T, 0, 1, 0',
	X =  -326.310  mm,	Y =    19.010  mm,	Z =     0.001  mm,
	W =  -167.366 deg,	P =    -0.002 deg,	R =   -78.266 deg
};
P[1925]{
   GP1:
	UF : 7, UT : 3,	CONFIG : 'F U T, 0, 1, 0',
	X =  -326.881  mm,	Y =     0.000  mm,	Z =     0.000  mm,
	W =  -167.362 deg,	P =     0.006 deg,	R =   -75.594 deg
};
P[1926]{
   GP1:
	UF : 7, UT : 3,	CONFIG : 'F U T, 0, 1, 0',
	X =  -326.881  mm,	Y =     0.000  mm,	Z =     0.000  mm,
	W =  -167.362 deg,	P =     0.006 deg,	R =   -75.594 deg
};
P[1927]{
   GP1:
	UF : 7, UT : 3,	CONFIG : 'F U T, 0, 1, 0',
	X =  -326.881  mm,	Y =     0.000  mm,	Z =     0.000  mm,
	W =  -167.362 deg,	P =     0.006 deg,	R =   -75.594 deg
};
P[1928]{
   GP1:
	UF : 7, UT : 3,	CONFIG : 'F U T, 0, 1, 0',
	X =  -326.881  mm,	Y =     0.000  mm,	Z =     0.000  mm,
	W =  -167.362 deg,	P =     0.006 deg,	R =   -75.594 deg
};
P[1929]{
   GP1:
	UF : 7, UT : 3,	CONFIG : 'F U T, 0, 1, 0',
	X =  -323.747  mm,	Y =     0.000  mm,	Z =     0.000  mm,
	W =  -167.362 deg,	P =     0.006 deg,	R =   -75.608 deg
};
P[1930]{
   GP1:
	UF : 7, UT : 3,	CONFIG : 'F U T, 0, 1, 0',
	X =  -323.747  mm,	Y =     0.000  mm,	Z =     0.000  mm,
	W =  -167.362 deg,	P =     0.006 deg,	R =   -75.608 deg
};
P[1931]{
   GP1:
	UF : 7, UT : 3,	CONFIG : 'F U T, 0, 1, 0',
	X =  -323.747  mm,	Y =     0.000  mm,	Z =     0.000  mm,
	W =  -167.362 deg,	P =     0.006 deg,	R =   -75.608 deg
};
P[1932]{
   GP1:
	UF : 7, UT : 3,	CONFIG : 'F U T, 0, 1, 0',
	X =  -323.747  mm,	Y =     0.000  mm,	Z =     0.000  mm,
	W =  -167.362 deg,	P =     0.006 deg,	R =   -75.608 deg
};
P[1933]{
   GP1:
	UF : 7, UT : 3,	CONFIG : 'F U T, 0, 1, 0',
	X =  -323.238  mm,	Y =    17.785  mm,	Z =     0.001  mm,
	W =  -167.365 deg,	P =    -0.002 deg,	R =   -78.103 deg
};
P[1934]{
   GP1:
	UF : 7, UT : 3,	CONFIG : 'F U T, 0, 1, 0',
	X =  -321.754  mm,	Y =    35.852  mm,	Z =     0.000  mm,
	W =  -167.367 deg,	P =    -0.010 deg,	R =   -80.713 deg
};
P[1935]{
   GP1:
	UF : 7, UT : 3,	CONFIG : 'F U T, 0, 1, 0',
	X =  -321.754  mm,	Y =    35.852  mm,	Z =     0.000  mm,
	W =  -167.367 deg,	P =    -0.010 deg,	R =   -80.713 deg
};
P[1936]{
   GP1:
	UF : 7, UT : 3,	CONFIG : 'F U T, 0, 1, 0',
	X =  -321.754  mm,	Y =    35.852  mm,	Z =     0.000  mm,
	W =  -167.367 deg,	P =    -0.010 deg,	R =   -80.713 deg
};
P[1937]{
   GP1:
	UF : 7, UT : 3,	CONFIG : 'F U T, 0, 1, 0',
	X =  -321.754  mm,	Y =    35.852  mm,	Z =     0.000  mm,
	W =  -167.367 deg,	P =    -0.010 deg,	R =   -80.713 deg
};
P[1938]{
   GP1:
	UF : 7, UT : 3,	CONFIG : 'F U T, 0, 0, 0',
	X =  -305.432  mm,	Y =   107.299  mm,	Z =     0.000  mm,
	W =  -167.234 deg,	P =     0.730 deg,	R =   -94.430 deg
};
P[1939]{
   GP1:
	UF : 7, UT : 3,	CONFIG : 'F U T, 0, 0, 0',
	X =  -305.432  mm,	Y =   107.299  mm,	Z =     0.000  mm,
	W =  -167.234 deg,	P =     0.730 deg,	R =   -94.430 deg
};
P[1940]{
   GP1:
	UF : 7, UT : 3,	CONFIG : 'F U T, 0, 0, 0',
	X =  -305.432  mm,	Y =   107.299  mm,	Z =     0.000  mm,
	W =  -167.234 deg,	P =     0.730 deg,	R =   -94.430 deg
};
P[1941]{
   GP1:
	UF : 7, UT : 3,	CONFIG : 'F U T, 0, 0, 0',
	X =  -305.432  mm,	Y =   107.299  mm,	Z =     0.000  mm,
	W =  -167.234 deg,	P =     0.730 deg,	R =   -94.430 deg
};
P[1942]{
   GP1:
	UF : 7, UT : 3,	CONFIG : 'F U T, 0, 0, 0',
	X =  -302.125  mm,	Y =   116.280  mm,	Z =     0.199  mm,
	W =  -167.481 deg,	P =     1.601 deg,	R =   -95.948 deg
};
P[1943]{
   GP1:
	UF : 7, UT : 3,	CONFIG : 'F U T, 0, 0, 0',
	X =  -299.172  mm,	Y =   123.693  mm,	Z =     0.412  mm,
	W =  -167.914 deg,	P =     1.607 deg,	R =   -97.367 deg
};
P[1944]{
   GP1:
	UF : 7, UT : 3,	CONFIG : 'F U T, 0, 0, 0',
	X =  -295.016  mm,	Y =   133.322  mm,	Z =     0.593  mm,
	W =  -168.300 deg,	P =     0.781 deg,	R =   -99.286 deg
};
P[1945]{
   GP1:
	UF : 7, UT : 3,	CONFIG : 'F U T, 0, 0, 0',
	X =  -286.754  mm,	Y =   150.265  mm,	Z =     0.553  mm,
	W =  -168.422 deg,	P =    -0.535 deg,	R =  -102.586 deg
};
P[1946]{
   GP1:
	UF : 7, UT : 3,	CONFIG : 'F U T, 0, 0, 0',
	X =  -279.860  mm,	Y =   162.734  mm,	Z =     0.260  mm,
	W =  -168.144 deg,	P =    -1.256 deg,	R =  -105.066 deg
};
P[1947]{
   GP1:
	UF : 7, UT : 3,	CONFIG : 'F U T, 0, 0, 0',
	X =  -274.323  mm,	Y =   171.896  mm,	Z =     0.000  mm,
	W =  -167.782 deg,	P =    -1.173 deg,	R =  -107.470 deg
};
P[1948]{
   GP1:
	UF : 7, UT : 3,	CONFIG : 'F U T, 0, 0, 0',
	X =  -274.323  mm,	Y =   171.896  mm,	Z =     0.000  mm,
	W =  -167.782 deg,	P =    -1.173 deg,	R =  -107.470 deg
};
P[1949]{
   GP1:
	UF : 7, UT : 3,	CONFIG : 'F U T, 0, 0, 0',
	X =  -274.323  mm,	Y =   171.896  mm,	Z =     0.000  mm,
	W =  -167.782 deg,	P =    -1.173 deg,	R =  -107.470 deg
};
P[1950]{
   GP1:
	UF : 7, UT : 3,	CONFIG : 'F U T, 0, 0, 0',
	X =  -274.323  mm,	Y =   171.896  mm,	Z =     0.000  mm,
	W =  -167.782 deg,	P =    -1.173 deg,	R =  -107.470 deg
};
P[1951]{
   GP1:
	UF : 7, UT : 3,	CONFIG : 'F U T, 0, 0, 0',
	X =  -228.627  mm,	Y =   229.192  mm,	Z =     0.000  mm,
	W =  -167.342 deg,	P =     0.116 deg,	R =  -119.428 deg
};
P[1952]{
   GP1:
	UF : 7, UT : 3,	CONFIG : 'F U T, 0, 0, 0',
	X =  -228.627  mm,	Y =   229.192  mm,	Z =     0.000  mm,
	W =  -167.342 deg,	P =     0.116 deg,	R =  -119.428 deg
};
P[1953]{
   GP1:
	UF : 7, UT : 3,	CONFIG : 'F U T, 0, 0, 0',
	X =  -228.627  mm,	Y =   229.192  mm,	Z =     0.000  mm,
	W =  -167.342 deg,	P =     0.116 deg,	R =  -119.428 deg
};
P[1954]{
   GP1:
	UF : 7, UT : 3,	CONFIG : 'F U T, 0, 0, 0',
	X =  -228.627  mm,	Y =   229.192  mm,	Z =     0.000  mm,
	W =  -167.342 deg,	P =     0.116 deg,	R =  -119.428 deg
};
P[1955]{
   GP1:
	UF : 7, UT : 3,	CONFIG : 'F U T, 0, 0, 0',
	X =  -218.512  mm,	Y =   238.857  mm,	Z =     0.018  mm,
	W =  -167.350 deg,	P =     0.051 deg,	R =  -122.439 deg
};
P[1956]{
   GP1:
	UF : 7, UT : 3,	CONFIG : 'F U T, 0, 0, 0',
	X =  -207.113  mm,	Y =   248.808  mm,	Z =     0.020  mm,
	W =  -167.350 deg,	P =    -0.020 deg,	R =  -125.142 deg
};
P[1957]{
   GP1:
	UF : 7, UT : 3,	CONFIG : 'F U T, 0, 0, 0',
	X =  -189.791  mm,	Y =   262.260  mm,	Z =     0.009  mm,
	W =  -167.360 deg,	P =    -0.017 deg,	R =  -128.976 deg
};
P[1958]{
   GP1:
	UF : 7, UT : 3,	CONFIG : 'F U T, 0, 0, 0',
	X =  -172.572  mm,	Y =   273.895  mm,	Z =     0.000  mm,
	W =  -167.369 deg,	P =    -0.016 deg,	R =  -133.028 deg
};
P[1959]{
   GP1:
	UF : 7, UT : 3,	CONFIG : 'F U T, 0, 0, 0',
	X =  -172.572  mm,	Y =   273.895  mm,	Z =     0.000  mm,
	W =  -167.369 deg,	P =    -0.016 deg,	R =  -133.028 deg
};
P[1960]{
   GP1:
	UF : 7, UT : 3,	CONFIG : 'F U T, 0, 0, 0',
	X =  -172.572  mm,	Y =   273.895  mm,	Z =     0.000  mm,
	W =  -167.369 deg,	P =    -0.016 deg,	R =  -133.028 deg
};
P[1961]{
   GP1:
	UF : 7, UT : 3,	CONFIG : 'F U T, 0, 0, 0',
	X =  -172.572  mm,	Y =   273.895  mm,	Z =     0.000  mm,
	W =  -167.369 deg,	P =    -0.016 deg,	R =  -133.028 deg
};
P[1962]{
   GP1:
	UF : 7, UT : 3,	CONFIG : 'F U T, 0, 0, 0',
	X =  -106.546  mm,	Y =   305.701  mm,	Z =     0.000  mm,
	W =  -167.363 deg,	P =     0.004 deg,	R =  -145.845 deg
};
P[1963]{
   GP1:
	UF : 7, UT : 3,	CONFIG : 'F U T, 0, 0, 0',
	X =  -106.546  mm,	Y =   305.701  mm,	Z =     0.000  mm,
	W =  -167.363 deg,	P =     0.004 deg,	R =  -145.845 deg
};
P[1964]{
   GP1:
	UF : 7, UT : 3,	CONFIG : 'F U T, 0, 0, 0',
	X =  -106.546  mm,	Y =   305.701  mm,	Z =     0.000  mm,
	W =  -167.363 deg,	P =     0.004 deg,	R =  -145.845 deg
};
P[1965]{
   GP1:
	UF : 7, UT : 3,	CONFIG : 'F U T, 0, 0, 0',
	X =  -106.546  mm,	Y =   305.701  mm,	Z =     0.000  mm,
	W =  -167.363 deg,	P =     0.004 deg,	R =  -145.845 deg
};
P[1966]{
   GP1:
	UF : 7, UT : 3,	CONFIG : 'F U T, 0, 0, 0',
	X =   -89.894  mm,	Y =   310.999  mm,	Z =     0.001  mm,
	W =  -167.363 deg,	P =     0.003 deg,	R =  -148.908 deg
};
P[1967]{
   GP1:
	UF : 7, UT : 3,	CONFIG : 'F U T, 0, 0, 0',
	X =   -72.777  mm,	Y =   315.449  mm,	Z =     0.001  mm,
	W =  -167.364 deg,	P =     0.002 deg,	R =  -151.945 deg
};
P[1968]{
   GP1:
	UF : 7, UT : 3,	CONFIG : 'F U T, 0, 0, 0',
	X =   -55.829  mm,	Y =   318.885  mm,	Z =     0.000  mm,
	W =  -167.364 deg,	P =     0.000 deg,	R =  -155.053 deg
};
P[1969]{
   GP1:
	UF : 7, UT : 3,	CONFIG : 'F U T, 0, 0, 0',
	X =   -36.644  mm,	Y =   321.658  mm,	Z =     0.000  mm,
	W =  -167.364 deg,	P =    -0.001 deg,	R =  -157.950 deg
};
P[1970]{
   GP1:
	UF : 7, UT : 3,	CONFIG : 'F U T, 0, 0, 0',
	X =   -36.644  mm,	Y =   321.658  mm,	Z =     0.000  mm,
	W =  -167.364 deg,	P =    -0.001 deg,	R =  -157.950 deg
};
P[1971]{
   GP1:
	UF : 7, UT : 3,	CONFIG : 'F U T, 0, 0, 0',
	X =   -36.644  mm,	Y =   321.658  mm,	Z =     0.000  mm,
	W =  -167.364 deg,	P =    -0.001 deg,	R =  -157.950 deg
};
P[1972]{
   GP1:
	UF : 7, UT : 3,	CONFIG : 'F U T, 0, 0, 0',
	X =   -36.644  mm,	Y =   321.658  mm,	Z =     0.000  mm,
	W =  -167.364 deg,	P =    -0.001 deg,	R =  -157.950 deg
};
P[1973]{
   GP1:
	UF : 7, UT : 3,	CONFIG : 'F U T, 0, 0, 0',
	X =    36.644  mm,	Y =   321.658  mm,	Z =     0.000  mm,
	W =  -167.363 deg,	P =     0.000 deg,	R =  -171.928 deg
};
P[1974]{
   GP1:
	UF : 7, UT : 3,	CONFIG : 'F U T, 0, 0, 0',
	X =    36.644  mm,	Y =   321.658  mm,	Z =     0.000  mm,
	W =  -167.363 deg,	P =     0.000 deg,	R =  -171.928 deg
};
P[1975]{
   GP1:
	UF : 7, UT : 3,	CONFIG : 'F U T, 0, 0, 0',
	X =    36.644  mm,	Y =   321.658  mm,	Z =     0.000  mm,
	W =  -167.363 deg,	P =     0.000 deg,	R =  -171.928 deg
};
P[1976]{
   GP1:
	UF : 7, UT : 3,	CONFIG : 'F U T, 0, 0, 0',
	X =    36.644  mm,	Y =   321.658  mm,	Z =     0.000  mm,
	W =  -167.363 deg,	P =     0.000 deg,	R =  -171.928 deg
};
P[1977]{
   GP1:
	UF : 7, UT : 3,	CONFIG : 'F U T, 0, 0, 0',
	X =    56.062  mm,	Y =   318.845  mm,	Z =     0.000  mm,
	W =  -167.364 deg,	P =     0.000 deg,	R =  -174.895 deg
};
P[1978]{
   GP1:
	UF : 7, UT : 3,	CONFIG : 'F U T, 0, 0, 0',
	X =    73.001  mm,	Y =   315.396  mm,	Z =     0.000  mm,
	W =  -167.364 deg,	P =     0.000 deg,	R =  -177.981 deg
};
P[1979]{
   GP1:
	UF : 7, UT : 3,	CONFIG : 'F U T, 0, 0, 0',
	X =    89.891  mm,	Y =   311.000  mm,	Z =     0.000  mm,
	W =  -167.364 deg,	P =     0.000 deg,	R =   178.977 deg
};
P[1980]{
   GP1:
	UF : 7, UT : 3,	CONFIG : 'F U T, 0, 0, 0',
	X =   106.546  mm,	Y =   305.701  mm,	Z =     0.000  mm,
	W =  -167.364 deg,	P =    -0.001 deg,	R =   175.952 deg
};
P[1981]{
   GP1:
	UF : 7, UT : 3,	CONFIG : 'F U T, 0, 0, 0',
	X =   106.546  mm,	Y =   305.701  mm,	Z =     0.000  mm,
	W =  -167.364 deg,	P =    -0.001 deg,	R =   175.952 deg
};
P[1982]{
   GP1:
	UF : 7, UT : 3,	CONFIG : 'F U T, 0, 0, 0',
	X =   106.546  mm,	Y =   305.701  mm,	Z =     0.000  mm,
	W =  -167.364 deg,	P =    -0.001 deg,	R =   175.952 deg
};
P[1983]{
   GP1:
	UF : 7, UT : 3,	CONFIG : 'F U T, 0, 0, 0',
	X =   106.546  mm,	Y =   305.701  mm,	Z =     0.000  mm,
	W =  -167.364 deg,	P =    -0.001 deg,	R =   175.952 deg
};
P[1984]{
   GP1:
	UF : 7, UT : 3,	CONFIG : 'F U T, 0, 0, 0',
	X =   172.572  mm,	Y =   273.895  mm,	Z =     0.000  mm,
	W =  -167.363 deg,	P =     0.002 deg,	R =   163.224 deg
};
P[1985]{
   GP1:
	UF : 7, UT : 3,	CONFIG : 'F U T, 0, 0, 0',
	X =   172.572  mm,	Y =   273.895  mm,	Z =     0.000  mm,
	W =  -167.363 deg,	P =     0.002 deg,	R =   163.224 deg
};
P[1986]{
   GP1:
	UF : 7, UT : 3,	CONFIG : 'F U T, 0, 0, 0',
	X =   172.572  mm,	Y =   273.895  mm,	Z =     0.000  mm,
	W =  -167.363 deg,	P =     0.002 deg,	R =   163.224 deg
};
P[1987]{
   GP1:
	UF : 7, UT : 3,	CONFIG : 'F U T, 0, 0, 0',
	X =   172.572  mm,	Y =   273.895  mm,	Z =     0.000  mm,
	W =  -167.363 deg,	P =     0.002 deg,	R =   163.224 deg
};
P[1988]{
   GP1:
	UF : 7, UT : 3,	CONFIG : 'F U T, 0, 0, 0',
	X =   187.242  mm,	Y =   264.099  mm,	Z =     0.001  mm,
	W =  -167.364 deg,	P =     0.001 deg,	R =   159.733 deg
};
P[1989]{
   GP1:
	UF : 7, UT : 3,	CONFIG : 'F U T, 0, 0, 0',
	X =   202.010  mm,	Y =   252.966  mm,	Z =     0.001  mm,
	W =  -167.364 deg,	P =     0.000 deg,	R =   156.448 deg
};
P[1990]{
   GP1:
	UF : 7, UT : 3,	CONFIG : 'F U T, 0, 0, 0',
	X =   216.163  mm,	Y =   240.994  mm,	Z =     0.001  mm,
	W =  -167.364 deg,	P =    -0.001 deg,	R =   153.167 deg
};
P[1991]{
   GP1:
	UF : 7, UT : 3,	CONFIG : 'F U T, 0, 0, 0',
	X =   228.627  mm,	Y =   229.192  mm,	Z =     0.000  mm,
	W =  -167.364 deg,	P =    -0.002 deg,	R =   149.541 deg
};
P[1992]{
   GP1:
	UF : 7, UT : 3,	CONFIG : 'F U T, 0, 0, 0',
	X =   228.627  mm,	Y =   229.192  mm,	Z =     0.000  mm,
	W =  -167.364 deg,	P =    -0.002 deg,	R =   149.541 deg
};
P[1993]{
   GP1:
	UF : 7, UT : 3,	CONFIG : 'F U T, 0, 0, 0',
	X =   228.627  mm,	Y =   229.192  mm,	Z =     0.000  mm,
	W =  -167.364 deg,	P =    -0.002 deg,	R =   149.541 deg
};
P[1994]{
   GP1:
	UF : 7, UT : 3,	CONFIG : 'F U T, 0, 0, 0',
	X =   228.627  mm,	Y =   229.192  mm,	Z =     0.000  mm,
	W =  -167.364 deg,	P =    -0.002 deg,	R =   149.541 deg
};
P[1995]{
   GP1:
	UF : 7, UT : 3,	CONFIG : 'F U T, 0, 0, 0',
	X =   274.323  mm,	Y =   171.896  mm,	Z =     0.000  mm,
	W =  -167.363 deg,	P =     0.002 deg,	R =   137.482 deg
};
P[1996]{
   GP1:
	UF : 7, UT : 3,	CONFIG : 'F U T, 0, 0, 0',
	X =   274.323  mm,	Y =   171.896  mm,	Z =     0.000  mm,
	W =  -167.363 deg,	P =     0.002 deg,	R =   137.482 deg
};
P[1997]{
   GP1:
	UF : 7, UT : 3,	CONFIG : 'F U T, 0, 0, 0',
	X =   274.323  mm,	Y =   171.896  mm,	Z =     0.000  mm,
	W =  -167.363 deg,	P =     0.002 deg,	R =   137.482 deg
};
P[1998]{
   GP1:
	UF : 7, UT : 3,	CONFIG : 'F U T, 0, 0, 0',
	X =   274.323  mm,	Y =   171.896  mm,	Z =     0.000  mm,
	W =  -167.363 deg,	P =     0.002 deg,	R =   137.482 deg
};
P[1999]{
   GP1:
	UF : 7, UT : 3,	CONFIG : 'F U T, 0, 0, 0',
	X =   283.027  mm,	Y =   157.162  mm,	Z =     0.000  mm,
	W =  -167.364 deg,	P =     0.001 deg,	R =   134.074 deg
};
P[2000]{
   GP1:
	UF : 7, UT : 3,	CONFIG : 'F U T, 0, 0, 0',
	X =   291.437  mm,	Y =   140.946  mm,	Z =     0.001  mm,
	W =  -167.364 deg,	P =     0.000 deg,	R =   130.910 deg
};
P[2001]{
   GP1:
	UF : 7, UT : 3,	CONFIG : 'F U T, 0, 0, 0',
	X =   298.756  mm,	Y =   124.694  mm,	Z =     0.001  mm,
	W =  -167.364 deg,	P =    -0.001 deg,	R =   127.670 deg
};
P[2002]{
   GP1:
	UF : 7, UT : 3,	CONFIG : 'F U T, 0, 0, 0',
	X =   305.432  mm,	Y =   107.299  mm,	Z =     0.000  mm,
	W =  -167.364 deg,	P =    -0.003 deg,	R =   124.542 deg
};
P[2003]{
   GP1:
	UF : 7, UT : 3,	CONFIG : 'F U T, 0, 0, 0',
	X =   305.432  mm,	Y =   107.299  mm,	Z =     0.000  mm,
	W =  -167.364 deg,	P =    -0.003 deg,	R =   124.542 deg
};
P[2004]{
   GP1:
	UF : 7, UT : 3,	CONFIG : 'F U T, 0, 0, 0',
	X =   305.432  mm,	Y =   107.299  mm,	Z =     0.000  mm,
	W =  -167.364 deg,	P =    -0.003 deg,	R =   124.542 deg
};
P[2005]{
   GP1:
	UF : 7, UT : 3,	CONFIG : 'F U T, 0, 0, 0',
	X =   305.432  mm,	Y =   107.299  mm,	Z =     0.000  mm,
	W =  -167.364 deg,	P =    -0.003 deg,	R =   124.542 deg
};
P[2006]{
   GP1:
	UF : 7, UT : 3,	CONFIG : 'F U T, 0, 0, 0',
	X =   321.754  mm,	Y =    35.852  mm,	Z =     0.000  mm,
	W =  -167.363 deg,	P =     0.001 deg,	R =   110.827 deg
};
P[2007]{
   GP1:
	UF : 7, UT : 3,	CONFIG : 'F U T, 0, 0, 0',
	X =   321.754  mm,	Y =    35.852  mm,	Z =     0.000  mm,
	W =  -167.363 deg,	P =     0.001 deg,	R =   110.827 deg
};
P[2008]{
   GP1:
	UF : 7, UT : 3,	CONFIG : 'F U T, 0, 0, 0',
	X =   321.754  mm,	Y =    35.852  mm,	Z =     0.000  mm,
	W =  -167.363 deg,	P =     0.001 deg,	R =   110.827 deg
};
P[2009]{
   GP1:
	UF : 7, UT : 3,	CONFIG : 'F U T, 0, 0, 0',
	X =   321.754  mm,	Y =    35.852  mm,	Z =     0.000  mm,
	W =  -167.363 deg,	P =     0.001 deg,	R =   110.827 deg
};
P[2010]{
   GP1:
	UF : 7, UT : 3,	CONFIG : 'F U T, 0, 0, 0',
	X =   323.214  mm,	Y =    18.222  mm,	Z =     0.000  mm,
	W =  -167.364 deg,	P =     0.000 deg,	R =   108.254 deg
};
P[2011]{
   GP1:
	UF : 7, UT : 3,	CONFIG : 'F U T, 0, 0, 0',
	X =   323.747  mm,	Y =     0.000  mm,	Z =     0.000  mm,
	W =  -167.364 deg,	P =    -0.001 deg,	R =   105.693 deg
};
P[2012]{
   GP1:
	UF : 7, UT : 3,	CONFIG : 'F U T, 0, 0, 0',
	X =   323.747  mm,	Y =     0.000  mm,	Z =     0.000  mm,
	W =  -167.364 deg,	P =    -0.001 deg,	R =   105.693 deg
};
P[2013]{
   GP1:
	UF : 7, UT : 3,	CONFIG : 'F U T, 0, 0, 0',
	X =   323.747  mm,	Y =     0.000  mm,	Z =     0.000  mm,
	W =  -167.364 deg,	P =    -0.001 deg,	R =   105.693 deg
};
P[2014]{
   GP1:
	UF : 7, UT : 3,	CONFIG : 'F U T, 0, 0, 0',
	X =   323.747  mm,	Y =     0.000  mm,	Z =     0.000  mm,
	W =  -167.364 deg,	P =    -0.001 deg,	R =   105.693 deg
};
P[2015]{
   GP1:
	UF : 7, UT : 3,	CONFIG : 'F U T, 0, 0, 0',
	X =   320.613  mm,	Y =     0.000  mm,	Z =     0.000  mm,
	W =  -167.364 deg,	P =    -0.001 deg,	R =   105.685 deg
};
P[2016]{
   GP1:
	UF : 7, UT : 3,	CONFIG : 'F U T, 0, 0, 0',
	X =   320.613  mm,	Y =     0.000  mm,	Z =     0.000  mm,
	W =  -167.364 deg,	P =    -0.001 deg,	R =   105.685 deg
};
P[2017]{
   GP1:
	UF : 7, UT : 3,	CONFIG : 'F U T, 0, 0, 0',
	X =   320.613  mm,	Y =     0.000  mm,	Z =     0.000  mm,
	W =  -167.364 deg,	P =    -0.001 deg,	R =   105.685 deg
};
P[2018]{
   GP1:
	UF : 7, UT : 3,	CONFIG : 'F U T, 0, 0, 0',
	X =   320.613  mm,	Y =     0.000  mm,	Z =     0.000  mm,
	W =  -167.364 deg,	P =    -0.001 deg,	R =   105.685 deg
};
P[2019]{
   GP1:
	UF : 7, UT : 3,	CONFIG : 'F U T, 0, 0, 0',
	X =   320.087  mm,	Y =    18.011  mm,	Z =     0.000  mm,
	W =  -167.364 deg,	P =     0.000 deg,	R =   108.267 deg
};
P[2020]{
   GP1:
	UF : 7, UT : 3,	CONFIG : 'F U T, 0, 0, 0',
	X =   318.656  mm,	Y =    35.365  mm,	Z =     0.000  mm,
	W =  -167.363 deg,	P =     0.001 deg,	R =   110.739 deg
};
P[2021]{
   GP1:
	UF : 7, UT : 3,	CONFIG : 'F U T, 0, 0, 0',
	X =   318.656  mm,	Y =    35.365  mm,	Z =     0.000  mm,
	W =  -167.363 deg,	P =     0.001 deg,	R =   110.739 deg
};
P[2022]{
   GP1:
	UF : 7, UT : 3,	CONFIG : 'F U T, 0, 0, 0',
	X =   318.656  mm,	Y =    35.365  mm,	Z =     0.000  mm,
	W =  -167.363 deg,	P =     0.001 deg,	R =   110.739 deg
};
P[2023]{
   GP1:
	UF : 7, UT : 3,	CONFIG : 'F U T, 0, 0, 0',
	X =   318.656  mm,	Y =    35.365  mm,	Z =     0.000  mm,
	W =  -167.363 deg,	P =     0.001 deg,	R =   110.739 deg
};
P[2024]{
   GP1:
	UF : 7, UT : 3,	CONFIG : 'F U T, 0, 0, 0',
	X =   302.428  mm,	Y =   106.392  mm,	Z =     0.000  mm,
	W =  -167.364 deg,	P =    -0.003 deg,	R =   124.533 deg
};
P[2025]{
   GP1:
	UF : 7, UT : 3,	CONFIG : 'F U T, 0, 0, 0',
	X =   302.428  mm,	Y =   106.392  mm,	Z =     0.000  mm,
	W =  -167.364 deg,	P =    -0.003 deg,	R =   124.533 deg
};
P[2026]{
   GP1:
	UF : 7, UT : 3,	CONFIG : 'F U T, 0, 0, 0',
	X =   302.428  mm,	Y =   106.392  mm,	Z =     0.000  mm,
	W =  -167.364 deg,	P =    -0.003 deg,	R =   124.533 deg
};
P[2027]{
   GP1:
	UF : 7, UT : 3,	CONFIG : 'F U T, 0, 0, 0',
	X =   302.428  mm,	Y =   106.392  mm,	Z =     0.000  mm,
	W =  -167.364 deg,	P =    -0.003 deg,	R =   124.533 deg
};
P[2028]{
   GP1:
	UF : 7, UT : 3,	CONFIG : 'F U T, 0, 0, 0',
	X =   295.903  mm,	Y =   123.395  mm,	Z =     0.001  mm,
	W =  -167.364 deg,	P =    -0.001 deg,	R =   127.655 deg
};
P[2029]{
   GP1:
	UF : 7, UT : 3,	CONFIG : 'F U T, 0, 0, 0',
	X =   288.703  mm,	Y =   139.400  mm,	Z =     0.001  mm,
	W =  -167.364 deg,	P =     0.000 deg,	R =   130.888 deg
};
P[2030]{
   GP1:
	UF : 7, UT : 3,	CONFIG : 'F U T, 0, 0, 0',
	X =   280.382  mm,	Y =   155.467  mm,	Z =     0.001  mm,
	W =  -167.363 deg,	P =     0.001 deg,	R =   134.031 deg
};
P[2031]{
   GP1:
	UF : 7, UT : 3,	CONFIG : 'F U T, 0, 0, 0',
	X =   271.742  mm,	Y =   170.114  mm,	Z =     0.000  mm,
	W =  -167.363 deg,	P =     0.002 deg,	R =   137.396 deg
};
P[2032]{
   GP1:
	UF : 7, UT : 3,	CONFIG : 'F U T, 0, 0, 0',
	X =   271.742  mm,	Y =   170.114  mm,	Z =     0.000  mm,
	W =  -167.363 deg,	P =     0.002 deg,	R =   137.396 deg
};
P[2033]{
   GP1:
	UF : 7, UT : 3,	CONFIG : 'F U T, 0, 0, 0',
	X =   271.742  mm,	Y =   170.114  mm,	Z =     0.000  mm,
	W =  -167.363 deg,	P =     0.002 deg,	R =   137.396 deg
};
P[2034]{
   GP1:
	UF : 7, UT : 3,	CONFIG : 'F U T, 0, 0, 0',
	X =   271.742  mm,	Y =   170.114  mm,	Z =     0.000  mm,
	W =  -167.363 deg,	P =     0.002 deg,	R =   137.396 deg
};
P[2035]{
   GP1:
	UF : 7, UT : 3,	CONFIG : 'F U T, 0, 0, 0',
	X =   226.314  mm,	Y =   227.073  mm,	Z =     0.000  mm,
	W =  -167.364 deg,	P =    -0.003 deg,	R =   149.494 deg
};
P[2036]{
   GP1:
	UF : 7, UT : 3,	CONFIG : 'F U T, 0, 0, 0',
	X =   226.314  mm,	Y =   227.073  mm,	Z =     0.000  mm,
	W =  -167.364 deg,	P =    -0.003 deg,	R =   149.494 deg
};
P[2037]{
   GP1:
	UF : 7, UT : 3,	CONFIG : 'F U T, 0, 0, 0',
	X =   226.314  mm,	Y =   227.073  mm,	Z =     0.000  mm,
	W =  -167.364 deg,	P =    -0.003 deg,	R =   149.494 deg
};
P[2038]{
   GP1:
	UF : 7, UT : 3,	CONFIG : 'F U T, 0, 0, 0',
	X =   226.314  mm,	Y =   227.073  mm,	Z =     0.000  mm,
	W =  -167.364 deg,	P =    -0.003 deg,	R =   149.494 deg
};
P[2039]{
   GP1:
	UF : 7, UT : 3,	CONFIG : 'F U T, 0, 0, 0',
	X =   214.128  mm,	Y =   238.612  mm,	Z =     0.001  mm,
	W =  -167.364 deg,	P =    -0.002 deg,	R =   153.155 deg
};
P[2040]{
   GP1:
	UF : 7, UT : 3,	CONFIG : 'F U T, 0, 0, 0',
	X =   200.198  mm,	Y =   250.403  mm,	Z =     0.001  mm,
	W =  -167.364 deg,	P =     0.000 deg,	R =   156.441 deg
};
P[2041]{
   GP1:
	UF : 7, UT : 3,	CONFIG : 'F U T, 0, 0, 0',
	X =   185.601  mm,	Y =   261.424  mm,	Z =     0.001  mm,
	W =  -167.363 deg,	P =     0.001 deg,	R =   159.705 deg
};
P[2042]{
   GP1:
	UF : 7, UT : 3,	CONFIG : 'F U T, 0, 0, 0',
	X =   171.020  mm,	Y =   271.169  mm,	Z =     0.000  mm,
	W =  -167.363 deg,	P =     0.002 deg,	R =   163.111 deg
};
P[2043]{
   GP1:
	UF : 7, UT : 3,	CONFIG : 'F U T, 0, 0, 0',
	X =   171.020  mm,	Y =   271.169  mm,	Z =     0.000  mm,
	W =  -167.363 deg,	P =     0.002 deg,	R =   163.111 deg
};
P[2044]{
   GP1:
	UF : 7, UT : 3,	CONFIG : 'F U T, 0, 0, 0',
	X =   171.020  mm,	Y =   271.169  mm,	Z =     0.000  mm,
	W =  -167.363 deg,	P =     0.002 deg,	R =   163.111 deg
};
P[2045]{
   GP1:
	UF : 7, UT : 3,	CONFIG : 'F U T, 0, 0, 0',
	X =   171.020  mm,	Y =   271.169  mm,	Z =     0.000  mm,
	W =  -167.363 deg,	P =     0.002 deg,	R =   163.111 deg
};
P[2046]{
   GP1:
	UF : 7, UT : 3,	CONFIG : 'F U T, 0, 0, 0',
	X =   105.382  mm,	Y =   302.789  mm,	Z =     0.000  mm,
	W =  -167.364 deg,	P =    -0.001 deg,	R =   175.980 deg
};
P[2047]{
   GP1:
	UF : 7, UT : 3,	CONFIG : 'F U T, 0, 0, 0',
	X =   105.382  mm,	Y =   302.789  mm,	Z =     0.000  mm,
	W =  -167.364 deg,	P =    -0.001 deg,	R =   175.980 deg
};
P[2048]{
   GP1:
	UF : 7, UT : 3,	CONFIG : 'F U T, 0, 0, 0',
	X =   105.382  mm,	Y =   302.789  mm,	Z =     0.000  mm,
	W =  -167.364 deg,	P =    -0.001 deg,	R =   175.980 deg
};
P[2049]{
   GP1:
	UF : 7, UT : 3,	CONFIG : 'F U T, 0, 0, 0',
	X =   105.382  mm,	Y =   302.789  mm,	Z =     0.000  mm,
	W =  -167.364 deg,	P =    -0.001 deg,	R =   175.980 deg
};
P[2050]{
   GP1:
	UF : 7, UT : 3,	CONFIG : 'F U T, 0, 0, 0',
	X =    89.059  mm,	Y =   307.979  mm,	Z =     0.000  mm,
	W =  -167.364 deg,	P =     0.000 deg,	R =   179.023 deg
};
P[2051]{
   GP1:
	UF : 7, UT : 3,	CONFIG : 'F U T, 0, 0, 0',
	X =    72.208  mm,	Y =   312.362  mm,	Z =     0.000  mm,
	W =  -167.364 deg,	P =     0.000 deg,	R =  -177.970 deg
};
P[2052]{
   GP1:
	UF : 7, UT : 3,	CONFIG : 'F U T, 0, 0, 0',
	X =    55.598  mm,	Y =   315.746  mm,	Z =     0.000  mm,
	W =  -167.363 deg,	P =     0.000 deg,	R =  -174.901 deg
};
P[2053]{
   GP1:
	UF : 7, UT : 3,	CONFIG : 'F U T, 0, 0, 0',
	X =    36.429  mm,	Y =   318.526  mm,	Z =     0.000  mm,
	W =  -167.363 deg,	P =     0.001 deg,	R =  -171.927 deg
};
P[2054]{
   GP1:
	UF : 7, UT : 3,	CONFIG : 'F U T, 0, 0, 0',
	X =    36.429  mm,	Y =   318.526  mm,	Z =     0.000  mm,
	W =  -167.363 deg,	P =     0.001 deg,	R =  -171.927 deg
};
P[2055]{
   GP1:
	UF : 7, UT : 3,	CONFIG : 'F U T, 0, 0, 0',
	X =    36.429  mm,	Y =   318.526  mm,	Z =     0.000  mm,
	W =  -167.363 deg,	P =     0.001 deg,	R =  -171.927 deg
};
P[2056]{
   GP1:
	UF : 7, UT : 3,	CONFIG : 'F U T, 0, 0, 0',
	X =    36.429  mm,	Y =   318.526  mm,	Z =     0.000  mm,
	W =  -167.363 deg,	P =     0.001 deg,	R =  -171.927 deg
};
P[2057]{
   GP1:
	UF : 7, UT : 3,	CONFIG : 'F U T, 0, 0, 0',
	X =   -36.429  mm,	Y =   318.526  mm,	Z =     0.000  mm,
	W =  -167.364 deg,	P =    -0.001 deg,	R =  -157.992 deg
};
P[2058]{
   GP1:
	UF : 7, UT : 3,	CONFIG : 'F U T, 0, 0, 0',
	X =   -36.429  mm,	Y =   318.526  mm,	Z =     0.000  mm,
	W =  -167.364 deg,	P =    -0.001 deg,	R =  -157.992 deg
};
P[2059]{
   GP1:
	UF : 7, UT : 3,	CONFIG : 'F U T, 0, 0, 0',
	X =   -36.429  mm,	Y =   318.526  mm,	Z =     0.000  mm,
	W =  -167.364 deg,	P =    -0.001 deg,	R =  -157.992 deg
};
P[2060]{
   GP1:
	UF : 7, UT : 3,	CONFIG : 'F U T, 0, 0, 0',
	X =   -36.429  mm,	Y =   318.526  mm,	Z =     0.000  mm,
	W =  -167.364 deg,	P =    -0.001 deg,	R =  -157.992 deg
};
P[2061]{
   GP1:
	UF : 7, UT : 3,	CONFIG : 'F U T, 0, 0, 0',
	X =   -55.427  mm,	Y =   315.774  mm,	Z =     0.000  mm,
	W =  -167.364 deg,	P =     0.000 deg,	R =  -155.025 deg
};
P[2062]{
   GP1:
	UF : 7, UT : 3,	CONFIG : 'F U T, 0, 0, 0',
	X =   -72.033  mm,	Y =   312.407  mm,	Z =     0.001  mm,
	W =  -167.363 deg,	P =     0.002 deg,	R =  -151.941 deg
};
P[2063]{
   GP1:
	UF : 7, UT : 3,	CONFIG : 'F U T, 0, 0, 0',
	X =   -88.851  mm,	Y =   308.037  mm,	Z =     0.001  mm,
	W =  -167.363 deg,	P =     0.003 deg,	R =  -148.939 deg
};
P[2064]{
   GP1:
	UF : 7, UT : 3,	CONFIG : 'F U T, 0, 0, 0',
	X =  -105.382  mm,	Y =   302.789  mm,	Z =     0.000  mm,
	W =  -167.362 deg,	P =     0.004 deg,	R =  -145.933 deg
};
P[2065]{
   GP1:
	UF : 7, UT : 3,	CONFIG : 'F U T, 0, 0, 0',
	X =  -105.382  mm,	Y =   302.789  mm,	Z =     0.000  mm,
	W =  -167.362 deg,	P =     0.004 deg,	R =  -145.933 deg
};
P[2066]{
   GP1:
	UF : 7, UT : 3,	CONFIG : 'F U T, 0, 0, 0',
	X =  -105.382  mm,	Y =   302.789  mm,	Z =     0.000  mm,
	W =  -167.362 deg,	P =     0.004 deg,	R =  -145.933 deg
};
P[2067]{
   GP1:
	UF : 7, UT : 3,	CONFIG : 'F U T, 0, 0, 0',
	X =  -105.382  mm,	Y =   302.789  mm,	Z =     0.000  mm,
	W =  -167.362 deg,	P =     0.004 deg,	R =  -145.933 deg
};
P[2068]{
   GP1:
	UF : 7, UT : 3,	CONFIG : 'F U T, 0, 0, 0',
	X =  -171.020  mm,	Y =   271.169  mm,	Z =     0.000  mm,
	W =  -167.368 deg,	P =    -0.018 deg,	R =  -133.025 deg
};
P[2069]{
   GP1:
	UF : 7, UT : 3,	CONFIG : 'F U T, 0, 0, 0',
	X =  -171.020  mm,	Y =   271.169  mm,	Z =     0.000  mm,
	W =  -167.368 deg,	P =    -0.018 deg,	R =  -133.025 deg
};
P[2070]{
   GP1:
	UF : 7, UT : 3,	CONFIG : 'F U T, 0, 0, 0',
	X =  -171.020  mm,	Y =   271.169  mm,	Z =     0.000  mm,
	W =  -167.368 deg,	P =    -0.018 deg,	R =  -133.025 deg
};
P[2071]{
   GP1:
	UF : 7, UT : 3,	CONFIG : 'F U T, 0, 0, 0',
	X =  -171.020  mm,	Y =   271.169  mm,	Z =     0.000  mm,
	W =  -167.368 deg,	P =    -0.018 deg,	R =  -133.025 deg
};
P[2072]{
   GP1:
	UF : 7, UT : 3,	CONFIG : 'F U T, 0, 0, 0',
	X =  -187.477  mm,	Y =   260.069  mm,	Z =     0.009  mm,
	W =  -167.358 deg,	P =    -0.020 deg,	R =  -129.098 deg
};
P[2073]{
   GP1:
	UF : 7, UT : 3,	CONFIG : 'F U T, 0, 0, 0',
	X =  -204.060  mm,	Y =   247.271  mm,	Z =     0.021  mm,
	W =  -167.348 deg,	P =    -0.023 deg,	R =  -125.372 deg
};
P[2074]{
   GP1:
	UF : 7, UT : 3,	CONFIG : 'F U T, 0, 0, 0',
	X =  -215.835  mm,	Y =   237.057  mm,	Z =     0.019  mm,
	W =  -167.343 deg,	P =     0.050 deg,	R =  -122.549 deg
};
P[2075]{
   GP1:
	UF : 7, UT : 3,	CONFIG : 'F U T, 0, 0, 0',
	X =  -226.314  mm,	Y =   227.073  mm,	Z =     0.000  mm,
	W =  -167.331 deg,	P =     0.117 deg,	R =  -119.398 deg
};
P[2076]{
   GP1:
	UF : 7, UT : 3,	CONFIG : 'F U T, 0, 0, 0',
	X =  -226.314  mm,	Y =   227.073  mm,	Z =     0.000  mm,
	W =  -167.331 deg,	P =     0.117 deg,	R =  -119.398 deg
};
P[2077]{
   GP1:
	UF : 7, UT : 3,	CONFIG : 'F U T, 0, 0, 0',
	X =  -226.314  mm,	Y =   227.073  mm,	Z =     0.000  mm,
	W =  -167.331 deg,	P =     0.117 deg,	R =  -119.398 deg
};
P[2078]{
   GP1:
	UF : 7, UT : 3,	CONFIG : 'F U T, 0, 0, 0',
	X =  -226.314  mm,	Y =   227.073  mm,	Z =     0.000  mm,
	W =  -167.331 deg,	P =     0.117 deg,	R =  -119.398 deg
};
P[2079]{
   GP1:
	UF : 7, UT : 3,	CONFIG : 'F U T, 0, 0, 0',
	X =  -271.742  mm,	Y =   170.114  mm,	Z =     0.000  mm,
	W =  -167.670 deg,	P =    -1.156 deg,	R =  -107.332 deg
};
P[2080]{
   GP1:
	UF : 7, UT : 3,	CONFIG : 'F U T, 0, 0, 0',
	X =  -271.742  mm,	Y =   170.114  mm,	Z =     0.000  mm,
	W =  -167.670 deg,	P =    -1.156 deg,	R =  -107.332 deg
};
P[2081]{
   GP1:
	UF : 7, UT : 3,	CONFIG : 'F U T, 0, 0, 0',
	X =  -271.742  mm,	Y =   170.114  mm,	Z =     0.000  mm,
	W =  -167.670 deg,	P =    -1.156 deg,	R =  -107.332 deg
};
P[2082]{
   GP1:
	UF : 7, UT : 3,	CONFIG : 'F U T, 0, 0, 0',
	X =  -271.742  mm,	Y =   170.114  mm,	Z =     0.000  mm,
	W =  -167.670 deg,	P =    -1.156 deg,	R =  -107.332 deg
};
P[2083]{
   GP1:
	UF : 7, UT : 3,	CONFIG : 'F U T, 0, 0, 0',
	X =  -274.706  mm,	Y =   165.277  mm,	Z =     0.127  mm,
	W =  -167.871 deg,	P =    -1.256 deg,	R =  -106.025 deg
};
P[2084]{
   GP1:
	UF : 7, UT : 3,	CONFIG : 'F U T, 0, 0, 0',
	X =  -281.744  mm,	Y =   152.978  mm,	Z =     0.434  mm,
	W =  -168.275 deg,	P =    -0.791 deg,	R =  -103.504 deg
};
P[2085]{
   GP1:
	UF : 7, UT : 3,	CONFIG : 'F U T, 0, 0, 0',
	X =  -290.413  mm,	Y =   135.821  mm,	Z =     0.560  mm,
	W =  -168.305 deg,	P =     0.505 deg,	R =  -100.002 deg
};
P[2086]{
   GP1:
	UF : 7, UT : 3,	CONFIG : 'F U T, 0, 0, 0',
	X =  -295.433  mm,	Y =   124.518  mm,	Z =     0.411  mm,
	W =  -167.958 deg,	P =     1.369 deg,	R =   -97.800 deg
};
P[2087]{
   GP1:
	UF : 7, UT : 3,	CONFIG : 'F U T, 0, 0, 0',
	X =  -297.236  mm,	Y =   120.134  mm,	Z =     0.303  mm,
	W =  -167.702 deg,	P =     1.518 deg,	R =   -97.034 deg
};
P[2088]{
   GP1:
	UF : 7, UT : 3,	CONFIG : 'F U T, 0, 0, 0',
	X =  -300.508  mm,	Y =   111.723  mm,	Z =     0.091  mm,
	W =  -167.277 deg,	P =     1.178 deg,	R =   -95.358 deg
};
P[2089]{
   GP1:
	UF : 7, UT : 3,	CONFIG : 'F U T, 0, 0, 0',
	X =  -302.428  mm,	Y =   106.392  mm,	Z =     0.000  mm,
	W =  -167.189 deg,	P =     0.643 deg,	R =   -94.404 deg
};
P[2090]{
   GP1:
	UF : 7, UT : 3,	CONFIG : 'F U T, 0, 0, 0',
	X =  -302.428  mm,	Y =   106.392  mm,	Z =     0.000  mm,
	W =  -167.189 deg,	P =     0.643 deg,	R =   -94.404 deg
};
P[2091]{
   GP1:
	UF : 7, UT : 3,	CONFIG : 'F U T, 0, 0, 0',
	X =  -302.428  mm,	Y =   106.392  mm,	Z =     0.000  mm,
	W =  -167.189 deg,	P =     0.643 deg,	R =   -94.404 deg
};
P[2092]{
   GP1:
	UF : 7, UT : 3,	CONFIG : 'F U T, 0, 0, 0',
	X =  -302.428  mm,	Y =   106.392  mm,	Z =     0.000  mm,
	W =  -167.189 deg,	P =     0.643 deg,	R =   -94.404 deg
};
P[2093]{
   GP1:
	UF : 7, UT : 3,	CONFIG : 'F U T, 0, 1, 0',
	X =  -318.656  mm,	Y =    35.365  mm,	Z =     0.000  mm,
	W =  -167.366 deg,	P =    -0.010 deg,	R =   -80.642 deg
};
P[2094]{
   GP1:
	UF : 7, UT : 3,	CONFIG : 'F U T, 0, 1, 0',
	X =  -318.656  mm,	Y =    35.365  mm,	Z =     0.000  mm,
	W =  -167.366 deg,	P =    -0.010 deg,	R =   -80.642 deg
};
P[2095]{
   GP1:
	UF : 7, UT : 3,	CONFIG : 'F U T, 0, 1, 0',
	X =  -318.656  mm,	Y =    35.365  mm,	Z =     0.000  mm,
	W =  -167.366 deg,	P =    -0.010 deg,	R =   -80.642 deg
};
P[2096]{
   GP1:
	UF : 7, UT : 3,	CONFIG : 'F U T, 0, 1, 0',
	X =  -318.656  mm,	Y =    35.365  mm,	Z =     0.000  mm,
	W =  -167.366 deg,	P =    -0.010 deg,	R =   -80.642 deg
};
P[2097]{
   GP1:
	UF : 7, UT : 3,	CONFIG : 'F U T, 0, 1, 0',
	X =  -320.116  mm,	Y =    17.484  mm,	Z =     0.001  mm,
	W =  -167.364 deg,	P =    -0.002 deg,	R =   -78.090 deg
};
P[2098]{
   GP1:
	UF : 7, UT : 3,	CONFIG : 'F U T, 0, 1, 0',
	X =  -320.613  mm,	Y =     0.000  mm,	Z =     0.000  mm,
	W =  -167.362 deg,	P =     0.006 deg,	R =   -75.605 deg
};
P[2099]{
   GP1:
	UF : 7, UT : 3,	CONFIG : 'F U T, 0, 1, 0',
	X =  -320.613  mm,	Y =     0.000  mm,	Z =     0.000  mm,
	W =  -167.362 deg,	P =     0.006 deg,	R =   -75.605 deg
};
P[2100]{
   GP1:
	UF : 7, UT : 3,	CONFIG : 'F U T, 0, 1, 0',
	X =  -320.613  mm,	Y =     0.000  mm,	Z =     0.000  mm,
	W =  -167.362 deg,	P =     0.006 deg,	R =   -75.605 deg
};
P[2101]{
   GP1:
	UF : 7, UT : 3,	CONFIG : 'F U T, 0, 1, 0',
	X =  -320.613  mm,	Y =     0.000  mm,	Z =     0.000  mm,
	W =  -167.362 deg,	P =     0.006 deg,	R =   -75.605 deg
};
P[2102]{
   GP1:
	UF : 7, UT : 3,	CONFIG : 'F U T, 0, 1, 0',
	X =  -317.478  mm,	Y =     0.000  mm,	Z =     0.000  mm,
	W =  -167.362 deg,	P =     0.006 deg,	R =   -75.593 deg
};
P[2103]{
   GP1:
	UF : 7, UT : 3,	CONFIG : 'F U T, 0, 1, 0',
	X =  -317.478  mm,	Y =     0.000  mm,	Z =     0.000  mm,
	W =  -167.362 deg,	P =     0.006 deg,	R =   -75.593 deg
};
P[2104]{
   GP1:
	UF : 7, UT : 3,	CONFIG : 'F U T, 0, 1, 0',
	X =  -317.478  mm,	Y =     0.000  mm,	Z =     0.000  mm,
	W =  -167.362 deg,	P =     0.006 deg,	R =   -75.593 deg
};
P[2105]{
   GP1:
	UF : 7, UT : 3,	CONFIG : 'F U T, 0, 1, 0',
	X =  -317.478  mm,	Y =     0.000  mm,	Z =     0.000  mm,
	W =  -167.362 deg,	P =     0.006 deg,	R =   -75.593 deg
};
P[2106]{
   GP1:
	UF : 7, UT : 3,	CONFIG : 'F U T, 0, 1, 0',
	X =  -316.965  mm,	Y =    17.696  mm,	Z =     0.001  mm,
	W =  -167.364 deg,	P =    -0.002 deg,	R =   -78.136 deg
};
P[2107]{
   GP1:
	UF : 7, UT : 3,	CONFIG : 'F U T, 0, 1, 0',
	X =  -315.526  mm,	Y =    35.143  mm,	Z =     0.000  mm,
	W =  -167.365 deg,	P =    -0.010 deg,	R =   -80.713 deg
};
P[2108]{
   GP1:
	UF : 7, UT : 3,	CONFIG : 'F U T, 0, 1, 0',
	X =  -315.526  mm,	Y =    35.143  mm,	Z =     0.000  mm,
	W =  -167.365 deg,	P =    -0.010 deg,	R =   -80.713 deg
};
P[2109]{
   GP1:
	UF : 7, UT : 3,	CONFIG : 'F U T, 0, 1, 0',
	X =  -315.526  mm,	Y =    35.143  mm,	Z =     0.000  mm,
	W =  -167.365 deg,	P =    -0.010 deg,	R =   -80.713 deg
};
P[2110]{
   GP1:
	UF : 7, UT : 3,	CONFIG : 'F U T, 0, 1, 0',
	X =  -315.526  mm,	Y =    35.143  mm,	Z =     0.000  mm,
	W =  -167.365 deg,	P =    -0.010 deg,	R =   -80.713 deg
};
P[2111]{
   GP1:
	UF : 7, UT : 3,	CONFIG : 'F U T, 0, 0, 0',
	X =  -299.514  mm,	Y =   105.233  mm,	Z =     0.000  mm,
	W =  -167.165 deg,	P =     0.551 deg,	R =   -94.443 deg
};
P[2112]{
   GP1:
	UF : 7, UT : 3,	CONFIG : 'F U T, 0, 0, 0',
	X =  -299.514  mm,	Y =   105.233  mm,	Z =     0.000  mm,
	W =  -167.165 deg,	P =     0.551 deg,	R =   -94.443 deg
};
P[2113]{
   GP1:
	UF : 7, UT : 3,	CONFIG : 'F U T, 0, 0, 0',
	X =  -299.514  mm,	Y =   105.233  mm,	Z =     0.000  mm,
	W =  -167.165 deg,	P =     0.551 deg,	R =   -94.443 deg
};
P[2114]{
   GP1:
	UF : 7, UT : 3,	CONFIG : 'F U T, 0, 0, 0',
	X =  -299.514  mm,	Y =   105.233  mm,	Z =     0.000  mm,
	W =  -167.165 deg,	P =     0.551 deg,	R =   -94.443 deg
};
P[2115]{
   GP1:
	UF : 7, UT : 3,	CONFIG : 'F U T, 0, 0, 0',
	X =  -295.965  mm,	Y =   114.849  mm,	Z =     0.171  mm,
	W =  -167.419 deg,	P =     1.267 deg,	R =   -96.127 deg
};
P[2116]{
   GP1:
	UF : 7, UT : 3,	CONFIG : 'F U T, 0, 0, 0',
	X =  -292.426  mm,	Y =   123.583  mm,	Z =     0.368  mm,
	W =  -167.902 deg,	P =     1.232 deg,	R =   -97.868 deg
};
P[2117]{
   GP1:
	UF : 7, UT : 3,	CONFIG : 'F U T, 0, 0, 0',
	X =  -287.102  mm,	Y =   135.502  mm,	Z =     0.509  mm,
	W =  -168.257 deg,	P =     0.436 deg,	R =  -100.196 deg
};
P[2118]{
   GP1:
	UF : 7, UT : 3,	CONFIG : 'F U T, 0, 0, 0',
	X =  -278.803  mm,	Y =   151.825  mm,	Z =     0.393  mm,
	W =  -168.186 deg,	P =    -0.729 deg,	R =  -103.545 deg
};
P[2119]{
   GP1:
	UF : 7, UT : 3,	CONFIG : 'F U T, 0, 0, 0',
	X =  -271.898  mm,	Y =   163.865  mm,	Z =     0.115  mm,
	W =  -167.761 deg,	P =    -1.183 deg,	R =  -106.031 deg
};
P[2120]{
   GP1:
	UF : 7, UT : 3,	CONFIG : 'F U T, 0, 0, 0',
	X =  -269.018  mm,	Y =   168.557  mm,	Z =     0.000  mm,
	W =  -167.557 deg,	P =    -1.117 deg,	R =  -107.447 deg
};
P[2121]{
   GP1:
	UF : 7, UT : 3,	CONFIG : 'F U T, 0, 0, 0',
	X =  -269.018  mm,	Y =   168.557  mm,	Z =     0.000  mm,
	W =  -167.557 deg,	P =    -1.117 deg,	R =  -107.447 deg
};
P[2122]{
   GP1:
	UF : 7, UT : 3,	CONFIG : 'F U T, 0, 0, 0',
	X =  -269.018  mm,	Y =   168.557  mm,	Z =     0.000  mm,
	W =  -167.557 deg,	P =    -1.117 deg,	R =  -107.447 deg
};
P[2123]{
   GP1:
	UF : 7, UT : 3,	CONFIG : 'F U T, 0, 0, 0',
	X =  -269.018  mm,	Y =   168.557  mm,	Z =     0.000  mm,
	W =  -167.557 deg,	P =    -1.117 deg,	R =  -107.447 deg
};
P[2124]{
   GP1:
	UF : 7, UT : 3,	CONFIG : 'F U T, 0, 0, 0',
	X =  -224.191  mm,	Y =   224.763  mm,	Z =     0.000  mm,
	W =  -167.319 deg,	P =     0.118 deg,	R =  -119.376 deg
};
P[2125]{
   GP1:
	UF : 7, UT : 3,	CONFIG : 'F U T, 0, 0, 0',
	X =  -224.191  mm,	Y =   224.763  mm,	Z =     0.000  mm,
	W =  -167.319 deg,	P =     0.118 deg,	R =  -119.376 deg
};
P[2126]{
   GP1:
	UF : 7, UT : 3,	CONFIG : 'F U T, 0, 0, 0',
	X =  -224.191  mm,	Y =   224.763  mm,	Z =     0.000  mm,
	W =  -167.319 deg,	P =     0.118 deg,	R =  -119.376 deg
};
P[2127]{
   GP1:
	UF : 7, UT : 3,	CONFIG : 'F U T, 0, 0, 0',
	X =  -224.191  mm,	Y =   224.763  mm,	Z =     0.000  mm,
	W =  -167.319 deg,	P =     0.118 deg,	R =  -119.376 deg
};
P[2128]{
   GP1:
	UF : 7, UT : 3,	CONFIG : 'F U T, 0, 0, 0',
	X =  -213.288  mm,	Y =   235.139  mm,	Z =     0.021  mm,
	W =  -167.336 deg,	P =     0.049 deg,	R =  -122.667 deg
};
P[2129]{
   GP1:
	UF : 7, UT : 3,	CONFIG : 'F U T, 0, 0, 0',
	X =  -201.094  mm,	Y =   245.657  mm,	Z =     0.021  mm,
	W =  -167.345 deg,	P =    -0.027 deg,	R =  -125.638 deg
};
P[2130]{
   GP1:
	UF : 7, UT : 3,	CONFIG : 'F U T, 0, 0, 0',
	X =  -185.106  mm,	Y =   257.920  mm,	Z =     0.010  mm,
	W =  -167.356 deg,	P =    -0.023 deg,	R =  -129.232 deg
};
P[2131]{
   GP1:
	UF : 7, UT : 3,	CONFIG : 'F U T, 0, 0, 0',
	X =  -169.241  mm,	Y =   268.585  mm,	Z =     0.000  mm,
	W =  -167.367 deg,	P =    -0.020 deg,	R =  -133.004 deg
};
P[2132]{
   GP1:
	UF : 7, UT : 3,	CONFIG : 'F U T, 0, 0, 0',
	X =  -169.241  mm,	Y =   268.585  mm,	Z =     0.000  mm,
	W =  -167.367 deg,	P =    -0.020 deg,	R =  -133.004 deg
};
P[2133]{
   GP1:
	UF : 7, UT : 3,	CONFIG : 'F U T, 0, 0, 0',
	X =  -169.241  mm,	Y =   268.585  mm,	Z =     0.000  mm,
	W =  -167.367 deg,	P =    -0.020 deg,	R =  -133.004 deg
};
P[2134]{
   GP1:
	UF : 7, UT : 3,	CONFIG : 'F U T, 0, 0, 0',
	X =  -169.241  mm,	Y =   268.585  mm,	Z =     0.000  mm,
	W =  -167.367 deg,	P =    -0.020 deg,	R =  -133.004 deg
};
P[2135]{
   GP1:
	UF : 7, UT : 3,	CONFIG : 'F U T, 0, 0, 0',
	X =  -104.470  mm,	Y =   299.786  mm,	Z =     0.000  mm,
	W =  -167.362 deg,	P =     0.004 deg,	R =  -145.854 deg
};
P[2136]{
   GP1:
	UF : 7, UT : 3,	CONFIG : 'F U T, 0, 0, 0',
	X =  -104.470  mm,	Y =   299.786  mm,	Z =     0.000  mm,
	W =  -167.362 deg,	P =     0.004 deg,	R =  -145.854 deg
};
P[2137]{
   GP1:
	UF : 7, UT : 3,	CONFIG : 'F U T, 0, 0, 0',
	X =  -104.470  mm,	Y =   299.786  mm,	Z =     0.000  mm,
	W =  -167.362 deg,	P =     0.004 deg,	R =  -145.854 deg
};
P[2138]{
   GP1:
	UF : 7, UT : 3,	CONFIG : 'F U T, 0, 0, 0',
	X =  -104.470  mm,	Y =   299.786  mm,	Z =     0.000  mm,
	W =  -167.362 deg,	P =     0.004 deg,	R =  -145.854 deg
};
P[2139]{
   GP1:
	UF : 7, UT : 3,	CONFIG : 'F U T, 0, 0, 0',
	X =   -82.656  mm,	Y =   306.518  mm,	Z =     0.001  mm,
	W =  -167.363 deg,	P =     0.002 deg,	R =  -149.878 deg
};
P[2140]{
   GP1:
	UF : 7, UT : 3,	CONFIG : 'F U T, 0, 0, 0',
	X =   -60.541  mm,	Y =   311.638  mm,	Z =     0.001  mm,
	W =  -167.363 deg,	P =     0.001 deg,	R =  -153.942 deg
};
P[2141]{
   GP1:
	UF : 7, UT : 3,	CONFIG : 'F U T, 0, 0, 0',
	X =   -35.948  mm,	Y =   315.428  mm,	Z =     0.000  mm,
	W =  -167.364 deg,	P =    -0.001 deg,	R =  -157.969 deg
};
P[2142]{
   GP1:
	UF : 7, UT : 3,	CONFIG : 'F U T, 0, 0, 0',
	X =   -35.948  mm,	Y =   315.428  mm,	Z =     0.000  mm,
	W =  -167.364 deg,	P =    -0.001 deg,	R =  -157.969 deg
};
P[2143]{
   GP1:
	UF : 7, UT : 3,	CONFIG : 'F U T, 0, 0, 0',
	X =   -35.948  mm,	Y =   315.428  mm,	Z =     0.000  mm,
	W =  -167.364 deg,	P =    -0.001 deg,	R =  -157.969 deg
};
P[2144]{
   GP1:
	UF : 7, UT : 3,	CONFIG : 'F U T, 0, 0, 0',
	X =   -35.948  mm,	Y =   315.428  mm,	Z =     0.000  mm,
	W =  -167.364 deg,	P =    -0.001 deg,	R =  -157.969 deg
};
P[2145]{
   GP1:
	UF : 7, UT : 3,	CONFIG : 'F U T, 0, 0, 0',
	X =    35.948  mm,	Y =   315.428  mm,	Z =     0.000  mm,
	W =  -167.363 deg,	P =     0.001 deg,	R =  -171.926 deg
};
P[2146]{
   GP1:
	UF : 7, UT : 3,	CONFIG : 'F U T, 0, 0, 0',
	X =    35.948  mm,	Y =   315.428  mm,	Z =     0.000  mm,
	W =  -167.363 deg,	P =     0.001 deg,	R =  -171.926 deg
};
P[2147]{
   GP1:
	UF : 7, UT : 3,	CONFIG : 'F U T, 0, 0, 0',
	X =    35.948  mm,	Y =   315.428  mm,	Z =     0.000  mm,
	W =  -167.363 deg,	P =     0.001 deg,	R =  -171.926 deg
};
P[2148]{
   GP1:
	UF : 7, UT : 3,	CONFIG : 'F U T, 0, 0, 0',
	X =    35.948  mm,	Y =   315.428  mm,	Z =     0.000  mm,
	W =  -167.363 deg,	P =     0.001 deg,	R =  -171.926 deg
};
P[2149]{
   GP1:
	UF : 7, UT : 3,	CONFIG : 'F U T, 0, 0, 0',
	X =    60.517  mm,	Y =   311.643  mm,	Z =     0.000  mm,
	W =  -167.363 deg,	P =     0.000 deg,	R =  -175.940 deg
};
P[2150]{
   GP1:
	UF : 7, UT : 3,	CONFIG : 'F U T, 0, 0, 0',
	X =    82.692  mm,	Y =   306.509  mm,	Z =     0.000  mm,
	W =  -167.364 deg,	P =     0.000 deg,	R =  -179.999 deg
};
P[2151]{
   GP1:
	UF : 7, UT : 3,	CONFIG : 'F U T, 0, 0, 0',
	X =   104.470  mm,	Y =   299.786  mm,	Z =     0.000  mm,
	W =  -167.364 deg,	P =    -0.001 deg,	R =   175.961 deg
};
P[2152]{
   GP1:
	UF : 7, UT : 3,	CONFIG : 'F U T, 0, 0, 0',
	X =   104.470  mm,	Y =   299.786  mm,	Z =     0.000  mm,
	W =  -167.364 deg,	P =    -0.001 deg,	R =   175.961 deg
};
P[2153]{
   GP1:
	UF : 7, UT : 3,	CONFIG : 'F U T, 0, 0, 0',
	X =   104.470  mm,	Y =   299.786  mm,	Z =     0.000  mm,
	W =  -167.364 deg,	P =    -0.001 deg,	R =   175.961 deg
};
P[2154]{
   GP1:
	UF : 7, UT : 3,	CONFIG : 'F U T, 0, 0, 0',
	X =   104.470  mm,	Y =   299.786  mm,	Z =     0.000  mm,
	W =  -167.364 deg,	P =    -0.001 deg,	R =   175.961 deg
};
P[2155]{
   GP1:
	UF : 7, UT : 3,	CONFIG : 'F U T, 0, 0, 0',
	X =   169.241  mm,	Y =   268.585  mm,	Z =     0.000  mm,
	W =  -167.363 deg,	P =     0.002 deg,	R =   163.143 deg
};
P[2156]{
   GP1:
	UF : 7, UT : 3,	CONFIG : 'F U T, 0, 0, 0',
	X =   169.241  mm,	Y =   268.585  mm,	Z =     0.000  mm,
	W =  -167.363 deg,	P =     0.002 deg,	R =   163.143 deg
};
P[2157]{
   GP1:
	UF : 7, UT : 3,	CONFIG : 'F U T, 0, 0, 0',
	X =   169.241  mm,	Y =   268.585  mm,	Z =     0.000  mm,
	W =  -167.363 deg,	P =     0.002 deg,	R =   163.143 deg
};
P[2158]{
   GP1:
	UF : 7, UT : 3,	CONFIG : 'F U T, 0, 0, 0',
	X =   169.241  mm,	Y =   268.585  mm,	Z =     0.000  mm,
	W =  -167.363 deg,	P =     0.002 deg,	R =   163.143 deg
};
P[2159]{
   GP1:
	UF : 7, UT : 3,	CONFIG : 'F U T, 0, 0, 0',
	X =   183.720  mm,	Y =   258.920  mm,	Z =     0.001  mm,
	W =  -167.363 deg,	P =     0.001 deg,	R =   159.718 deg
};
P[2160]{
   GP1:
	UF : 7, UT : 3,	CONFIG : 'F U T, 0, 0, 0',
	X =   198.126  mm,	Y =   248.045  mm,	Z =     0.001  mm,
	W =  -167.364 deg,	P =     0.000 deg,	R =   156.405 deg
};
P[2161]{
   GP1:
	UF : 7, UT : 3,	CONFIG : 'F U T, 0, 0, 0',
	X =   212.090  mm,	Y =   236.233  mm,	Z =     0.001  mm,
	W =  -167.364 deg,	P =    -0.002 deg,	R =   153.153 deg
};
P[2162]{
   GP1:
	UF : 7, UT : 3,	CONFIG : 'F U T, 0, 0, 0',
	X =   224.191  mm,	Y =   224.763  mm,	Z =     0.000  mm,
	W =  -167.364 deg,	P =    -0.003 deg,	R =   149.479 deg
};
P[2163]{
   GP1:
	UF : 7, UT : 3,	CONFIG : 'F U T, 0, 0, 0',
	X =   224.191  mm,	Y =   224.763  mm,	Z =     0.000  mm,
	W =  -167.364 deg,	P =    -0.003 deg,	R =   149.479 deg
};
P[2164]{
   GP1:
	UF : 7, UT : 3,	CONFIG : 'F U T, 0, 0, 0',
	X =   224.191  mm,	Y =   224.763  mm,	Z =     0.000  mm,
	W =  -167.364 deg,	P =    -0.003 deg,	R =   149.479 deg
};
P[2165]{
   GP1:
	UF : 7, UT : 3,	CONFIG : 'F U T, 0, 0, 0',
	X =   224.191  mm,	Y =   224.763  mm,	Z =     0.000  mm,
	W =  -167.364 deg,	P =    -0.003 deg,	R =   149.479 deg
};
P[2166]{
   GP1:
	UF : 7, UT : 3,	CONFIG : 'F U T, 0, 0, 0',
	X =   269.018  mm,	Y =   168.557  mm,	Z =     0.000  mm,
	W =  -167.363 deg,	P =     0.003 deg,	R =   137.473 deg
};
P[2167]{
   GP1:
	UF : 7, UT : 3,	CONFIG : 'F U T, 0, 0, 0',
	X =   269.018  mm,	Y =   168.557  mm,	Z =     0.000  mm,
	W =  -167.363 deg,	P =     0.003 deg,	R =   137.473 deg
};
P[2168]{
   GP1:
	UF : 7, UT : 3,	CONFIG : 'F U T, 0, 0, 0',
	X =   269.018  mm,	Y =   168.557  mm,	Z =     0.000  mm,
	W =  -167.363 deg,	P =     0.003 deg,	R =   137.473 deg
};
P[2169]{
   GP1:
	UF : 7, UT : 3,	CONFIG : 'F U T, 0, 0, 0',
	X =   269.018  mm,	Y =   168.557  mm,	Z =     0.000  mm,
	W =  -167.363 deg,	P =     0.003 deg,	R =   137.473 deg
};
P[2170]{
   GP1:
	UF : 7, UT : 3,	CONFIG : 'F U T, 0, 0, 0',
	X =   277.589  mm,	Y =   154.047  mm,	Z =     0.001  mm,
	W =  -167.363 deg,	P =     0.001 deg,	R =   134.070 deg
};
P[2171]{
   GP1:
	UF : 7, UT : 3,	CONFIG : 'F U T, 0, 0, 0',
	X =   285.805  mm,	Y =   138.195  mm,	Z =     0.001  mm,
	W =  -167.364 deg,	P =     0.000 deg,	R =   130.902 deg
};
P[2172]{
   GP1:
	UF : 7, UT : 3,	CONFIG : 'F U T, 0, 0, 0',
	X =   292.963  mm,	Y =   122.300  mm,	Z =     0.001  mm,
	W =  -167.364 deg,	P =    -0.001 deg,	R =   127.666 deg
};
P[2173]{
   GP1:
	UF : 7, UT : 3,	CONFIG : 'F U T, 0, 0, 0',
	X =   299.514  mm,	Y =   105.233  mm,	Z =     0.000  mm,
	W =  -167.364 deg,	P =    -0.003 deg,	R =   124.545 deg
};
P[2174]{
   GP1:
	UF : 7, UT : 3,	CONFIG : 'F U T, 0, 0, 0',
	X =   299.514  mm,	Y =   105.233  mm,	Z =     0.000  mm,
	W =  -167.364 deg,	P =    -0.003 deg,	R =   124.545 deg
};
P[2175]{
   GP1:
	UF : 7, UT : 3,	CONFIG : 'F U T, 0, 0, 0',
	X =   299.514  mm,	Y =   105.233  mm,	Z =     0.000  mm,
	W =  -167.364 deg,	P =    -0.003 deg,	R =   124.545 deg
};
P[2176]{
   GP1:
	UF : 7, UT : 3,	CONFIG : 'F U T, 0, 0, 0',
	X =   299.514  mm,	Y =   105.233  mm,	Z =     0.000  mm,
	W =  -167.364 deg,	P =    -0.003 deg,	R =   124.545 deg
};
P[2177]{
   GP1:
	UF : 7, UT : 3,	CONFIG : 'F U T, 0, 0, 0',
	X =   315.526  mm,	Y =    35.143  mm,	Z =     0.000  mm,
	W =  -167.363 deg,	P =     0.001 deg,	R =   110.775 deg
};
P[2178]{
   GP1:
	UF : 7, UT : 3,	CONFIG : 'F U T, 0, 0, 0',
	X =   315.526  mm,	Y =    35.143  mm,	Z =     0.000  mm,
	W =  -167.363 deg,	P =     0.001 deg,	R =   110.775 deg
};
P[2179]{
   GP1:
	UF : 7, UT : 3,	CONFIG : 'F U T, 0, 0, 0',
	X =   315.526  mm,	Y =    35.143  mm,	Z =     0.000  mm,
	W =  -167.363 deg,	P =     0.001 deg,	R =   110.775 deg
};
P[2180]{
   GP1:
	UF : 7, UT : 3,	CONFIG : 'F U T, 0, 0, 0',
	X =   315.526  mm,	Y =    35.143  mm,	Z =     0.000  mm,
	W =  -167.363 deg,	P =     0.001 deg,	R =   110.775 deg
};
P[2181]{
   GP1:
	UF : 7, UT : 3,	CONFIG : 'F U T, 0, 0, 0',
	X =   316.958  mm,	Y =    17.828  mm,	Z =     0.000  mm,
	W =  -167.363 deg,	P =     0.000 deg,	R =   108.286 deg
};
P[2182]{
   GP1:
	UF : 7, UT : 3,	CONFIG : 'F U T, 0, 0, 0',
	X =   317.478  mm,	Y =     0.000  mm,	Z =     0.000  mm,
	W =  -167.364 deg,	P =    -0.001 deg,	R =   105.693 deg
};
P[2183]{
   GP1:
	UF : 7, UT : 3,	CONFIG : 'F U T, 0, 0, 0',
	X =   317.478  mm,	Y =     0.000  mm,	Z =     0.000  mm,
	W =  -167.364 deg,	P =    -0.001 deg,	R =   105.693 deg
};
P[2184]{
   GP1:
	UF : 7, UT : 3,	CONFIG : 'F U T, 0, 0, 0',
	X =   317.478  mm,	Y =     0.000  mm,	Z =     0.000  mm,
	W =  -167.364 deg,	P =    -0.001 deg,	R =   105.693 deg
};
P[2185]{
   GP1:
	UF : 7, UT : 3,	CONFIG : 'F U T, 0, 0, 0',
	X =   317.478  mm,	Y =     0.000  mm,	Z =     0.000  mm,
	W =  -167.364 deg,	P =    -0.001 deg,	R =   105.693 deg
};
P[2186]{
   GP1:
	UF : 7, UT : 3,	CONFIG : 'F U T, 0, 0, 0',
	X =   314.344  mm,	Y =     0.000  mm,	Z =     0.000  mm,
	W =  -167.364 deg,	P =    -0.001 deg,	R =   105.705 deg
};
P[2187]{
   GP1:
	UF : 7, UT : 3,	CONFIG : 'F U T, 0, 0, 0',
	X =   314.344  mm,	Y =     0.000  mm,	Z =     0.000  mm,
	W =  -167.364 deg,	P =    -0.001 deg,	R =   105.705 deg
};
P[2188]{
   GP1:
	UF : 7, UT : 3,	CONFIG : 'F U T, 0, 0, 0',
	X =   314.344  mm,	Y =     0.000  mm,	Z =     0.000  mm,
	W =  -167.364 deg,	P =    -0.001 deg,	R =   105.705 deg
};
P[2189]{
   GP1:
	UF : 7, UT : 3,	CONFIG : 'F U T, 0, 0, 0',
	X =   314.344  mm,	Y =     0.000  mm,	Z =     0.000  mm,
	W =  -167.364 deg,	P =    -0.001 deg,	R =   105.705 deg
};
P[2190]{
   GP1:
	UF : 7, UT : 3,	CONFIG : 'F U T, 0, 0, 0',
	X =   313.796  mm,	Y =    18.258  mm,	Z =     0.000  mm,
	W =  -167.363 deg,	P =     0.000 deg,	R =   108.359 deg
};
P[2191]{
   GP1:
	UF : 7, UT : 3,	CONFIG : 'F U T, 0, 0, 0',
	X =   312.363  mm,	Y =    35.193  mm,	Z =     0.000  mm,
	W =  -167.363 deg,	P =     0.001 deg,	R =   111.081 deg
};
P[2192]{
   GP1:
	UF : 7, UT : 3,	CONFIG : 'F U T, 0, 0, 0',
	X =   312.363  mm,	Y =    35.193  mm,	Z =     0.000  mm,
	W =  -167.363 deg,	P =     0.001 deg,	R =   111.081 deg
};
P[2193]{
   GP1:
	UF : 7, UT : 3,	CONFIG : 'F U T, 0, 0, 0',
	X =   312.363  mm,	Y =    35.193  mm,	Z =     0.000  mm,
	W =  -167.363 deg,	P =     0.001 deg,	R =   111.081 deg
};
P[2194]{
   GP1:
	UF : 7, UT : 3,	CONFIG : 'F U T, 0, 0, 0',
	X =   312.363  mm,	Y =    35.193  mm,	Z =     0.000  mm,
	W =  -167.363 deg,	P =     0.001 deg,	R =   111.081 deg
};
P[2195]{
   GP1:
	UF : 7, UT : 3,	CONFIG : 'F U T, 0, 0, 0',
	X =   296.692  mm,	Y =   103.818  mm,	Z =     0.000  mm,
	W =  -167.364 deg,	P =    -0.003 deg,	R =   124.612 deg
};
P[2196]{
   GP1:
	UF : 7, UT : 3,	CONFIG : 'F U T, 0, 0, 0',
	X =   296.692  mm,	Y =   103.818  mm,	Z =     0.000  mm,
	W =  -167.364 deg,	P =    -0.003 deg,	R =   124.612 deg
};
P[2197]{
   GP1:
	UF : 7, UT : 3,	CONFIG : 'F U T, 0, 0, 0',
	X =   296.692  mm,	Y =   103.818  mm,	Z =     0.000  mm,
	W =  -167.364 deg,	P =    -0.003 deg,	R =   124.612 deg
};
P[2198]{
   GP1:
	UF : 7, UT : 3,	CONFIG : 'F U T, 0, 0, 0',
	X =   296.692  mm,	Y =   103.818  mm,	Z =     0.000  mm,
	W =  -167.364 deg,	P =    -0.003 deg,	R =   124.612 deg
};
P[2199]{
   GP1:
	UF : 7, UT : 3,	CONFIG : 'F U T, 0, 0, 0',
	X =   289.976  mm,	Y =   121.319  mm,	Z =     0.001  mm,
	W =  -167.364 deg,	P =    -0.001 deg,	R =   127.739 deg
};
P[2200]{
   GP1:
	UF : 7, UT : 3,	CONFIG : 'F U T, 0, 0, 0',
	X =   282.724  mm,	Y =   137.365  mm,	Z =     0.001  mm,
	W =  -167.363 deg,	P =     0.000 deg,	R =   130.985 deg
};
P[2201]{
   GP1:
	UF : 7, UT : 3,	CONFIG : 'F U T, 0, 0, 0',
	X =   274.534  mm,	Y =   153.088  mm,	Z =     0.001  mm,
	W =  -167.363 deg,	P =     0.001 deg,	R =   134.198 deg
};
P[2202]{
   GP1:
	UF : 7, UT : 3,	CONFIG : 'F U T, 0, 0, 0',
	X =   266.148  mm,	Y =   167.232  mm,	Z =     0.000  mm,
	W =  -167.362 deg,	P =     0.003 deg,	R =   137.749 deg
};
P[2203]{
   GP1:
	UF : 7, UT : 3,	CONFIG : 'F U T, 0, 0, 0',
	X =   266.148  mm,	Y =   167.232  mm,	Z =     0.000  mm,
	W =  -167.362 deg,	P =     0.003 deg,	R =   137.749 deg
};
P[2204]{
   GP1:
	UF : 7, UT : 3,	CONFIG : 'F U T, 0, 0, 0',
	X =   266.148  mm,	Y =   167.232  mm,	Z =     0.000  mm,
	W =  -167.362 deg,	P =     0.003 deg,	R =   137.749 deg
};
P[2205]{
   GP1:
	UF : 7, UT : 3,	CONFIG : 'F U T, 0, 0, 0',
	X =   266.148  mm,	Y =   167.232  mm,	Z =     0.000  mm,
	W =  -167.362 deg,	P =     0.003 deg,	R =   137.749 deg
};
P[2206]{
   GP1:
	UF : 7, UT : 3,	CONFIG : 'F U T, 0, 0, 0',
	X =   222.261  mm,	Y =   222.261  mm,	Z =     0.000  mm,
	W =  -167.364 deg,	P =    -0.003 deg,	R =   149.599 deg
};
P[2207]{
   GP1:
	UF : 7, UT : 3,	CONFIG : 'F U T, 0, 0, 0',
	X =   222.261  mm,	Y =   222.261  mm,	Z =     0.000  mm,
	W =  -167.364 deg,	P =    -0.003 deg,	R =   149.599 deg
};
P[2208]{
   GP1:
	UF : 7, UT : 3,	CONFIG : 'F U T, 0, 0, 0',
	X =   222.261  mm,	Y =   222.261  mm,	Z =     0.000  mm,
	W =  -167.364 deg,	P =    -0.003 deg,	R =   149.599 deg
};
P[2209]{
   GP1:
	UF : 7, UT : 3,	CONFIG : 'F U T, 0, 0, 0',
	X =   222.261  mm,	Y =   222.261  mm,	Z =     0.000  mm,
	W =  -167.364 deg,	P =    -0.003 deg,	R =   149.599 deg
};
P[2210]{
   GP1:
	UF : 7, UT : 3,	CONFIG : 'F U T, 0, 0, 0',
	X =   209.897  mm,	Y =   233.994  mm,	Z =     0.001  mm,
	W =  -167.364 deg,	P =    -0.002 deg,	R =   153.153 deg
};
P[2211]{
   GP1:
	UF : 7, UT : 3,	CONFIG : 'F U T, 0, 0, 0',
	X =   195.899  mm,	Y =   245.814  mm,	Z =     0.001  mm,
	W =  -167.363 deg,	P =     0.000 deg,	R =   156.411 deg
};
P[2212]{
   GP1:
	UF : 7, UT : 3,	CONFIG : 'F U T, 0, 0, 0',
	X =   181.688  mm,	Y =   256.510  mm,	Z =     0.001  mm,
	W =  -167.363 deg,	P =     0.001 deg,	R =   159.771 deg
};
P[2213]{
   GP1:
	UF : 7, UT : 3,	CONFIG : 'F U T, 0, 0, 0',
	X =   167.232  mm,	Y =   266.148  mm,	Z =     0.000  mm,
	W =  -167.362 deg,	P =     0.002 deg,	R =   163.242 deg
};
P[2214]{
   GP1:
	UF : 7, UT : 3,	CONFIG : 'F U T, 0, 0, 0',
	X =   167.232  mm,	Y =   266.148  mm,	Z =     0.000  mm,
	W =  -167.362 deg,	P =     0.002 deg,	R =   163.242 deg
};
P[2215]{
   GP1:
	UF : 7, UT : 3,	CONFIG : 'F U T, 0, 0, 0',
	X =   167.232  mm,	Y =   266.148  mm,	Z =     0.000  mm,
	W =  -167.362 deg,	P =     0.002 deg,	R =   163.242 deg
};
P[2216]{
   GP1:
	UF : 7, UT : 3,	CONFIG : 'F U T, 0, 0, 0',
	X =   167.232  mm,	Y =   266.148  mm,	Z =     0.000  mm,
	W =  -167.362 deg,	P =     0.002 deg,	R =   163.242 deg
};
P[2217]{
   GP1:
	UF : 7, UT : 3,	CONFIG : 'F U T, 0, 0, 0',
	X =   103.816  mm,	Y =   296.692  mm,	Z =     0.000  mm,
	W =  -167.364 deg,	P =    -0.001 deg,	R =   175.609 deg
};
P[2218]{
   GP1:
	UF : 7, UT : 3,	CONFIG : 'F U T, 0, 0, 0',
	X =   103.816  mm,	Y =   296.692  mm,	Z =     0.000  mm,
	W =  -167.364 deg,	P =    -0.001 deg,	R =   175.609 deg
};
P[2219]{
   GP1:
	UF : 7, UT : 3,	CONFIG : 'F U T, 0, 0, 0',
	X =   103.816  mm,	Y =   296.692  mm,	Z =     0.000  mm,
	W =  -167.364 deg,	P =    -0.001 deg,	R =   175.609 deg
};
P[2220]{
   GP1:
	UF : 7, UT : 3,	CONFIG : 'F U T, 0, 0, 0',
	X =   103.816  mm,	Y =   296.692  mm,	Z =     0.000  mm,
	W =  -167.364 deg,	P =    -0.001 deg,	R =   175.609 deg
};
P[2221]{
   GP1:
	UF : 7, UT : 3,	CONFIG : 'F U T, 0, 0, 0',
	X =    87.953  mm,	Y =   301.775  mm,	Z =     0.000  mm,
	W =  -167.364 deg,	P =    -0.001 deg,	R =   178.852 deg
};
P[2222]{
   GP1:
	UF : 7, UT : 3,	CONFIG : 'F U T, 0, 0, 0',
	X =    71.164  mm,	Y =   306.169  mm,	Z =     0.000  mm,
	W =  -167.363 deg,	P =     0.000 deg,	R =  -178.042 deg
};
P[2223]{
   GP1:
	UF : 7, UT : 3,	CONFIG : 'F U T, 0, 0, 0',
	X =    54.389  mm,	Y =   309.594  mm,	Z =     0.000  mm,
	W =  -167.363 deg,	P =     0.000 deg,	R =  -174.890 deg
};
P[2224]{
   GP1:
	UF : 7, UT : 3,	CONFIG : 'F U T, 0, 0, 0',
	X =    35.197  mm,	Y =   312.362  mm,	Z =     0.000  mm,
	W =  -167.363 deg,	P =     0.001 deg,	R =  -171.894 deg
};
P[2225]{
   GP1:
	UF : 7, UT : 3,	CONFIG : 'F U T, 0, 0, 0',
	X =    35.197  mm,	Y =   312.362  mm,	Z =     0.000  mm,
	W =  -167.363 deg,	P =     0.001 deg,	R =  -171.894 deg
};
P[2226]{
   GP1:
	UF : 7, UT : 3,	CONFIG : 'F U T, 0, 0, 0',
	X =    35.197  mm,	Y =   312.362  mm,	Z =     0.000  mm,
	W =  -167.363 deg,	P =     0.001 deg,	R =  -171.894 deg
};
P[2227]{
   GP1:
	UF : 7, UT : 3,	CONFIG : 'F U T, 0, 0, 0',
	X =    35.197  mm,	Y =   312.362  mm,	Z =     0.000  mm,
	W =  -167.363 deg,	P =     0.001 deg,	R =  -171.894 deg
};
P[2228]{
   GP1:
	UF : 7, UT : 3,	CONFIG : 'F U T, 0, 0, 0',
	X =   -35.197  mm,	Y =   312.362  mm,	Z =     0.000  mm,
	W =  -167.364 deg,	P =    -0.001 deg,	R =  -157.993 deg
};
P[2229]{
   GP1:
	UF : 7, UT : 3,	CONFIG : 'F U T, 0, 0, 0',
	X =   -35.197  mm,	Y =   312.362  mm,	Z =     0.000  mm,
	W =  -167.364 deg,	P =    -0.001 deg,	R =  -157.993 deg
};
P[2230]{
   GP1:
	UF : 7, UT : 3,	CONFIG : 'F U T, 0, 0, 0',
	X =   -35.197  mm,	Y =   312.362  mm,	Z =     0.000  mm,
	W =  -167.364 deg,	P =    -0.001 deg,	R =  -157.993 deg
};
P[2231]{
   GP1:
	UF : 7, UT : 3,	CONFIG : 'F U T, 0, 0, 0',
	X =   -35.197  mm,	Y =   312.362  mm,	Z =     0.000  mm,
	W =  -167.364 deg,	P =    -0.001 deg,	R =  -157.993 deg
};
P[2232]{
   GP1:
	UF : 7, UT : 3,	CONFIG : 'F U T, 0, 0, 0',
	X =   -54.397  mm,	Y =   309.592  mm,	Z =     0.001  mm,
	W =  -167.363 deg,	P =     0.000 deg,	R =  -154.999 deg
};
P[2233]{
   GP1:
	UF : 7, UT : 3,	CONFIG : 'F U T, 0, 0, 0',
	X =   -71.123  mm,	Y =   306.179  mm,	Z =     0.001  mm,
	W =  -167.363 deg,	P =     0.002 deg,	R =  -151.872 deg
};
P[2234]{
   GP1:
	UF : 7, UT : 3,	CONFIG : 'F U T, 0, 0, 0',
	X =   -87.830  mm,	Y =   301.810  mm,	Z =     0.001  mm,
	W =  -167.362 deg,	P =     0.003 deg,	R =  -148.771 deg
};
P[2235]{
   GP1:
	UF : 7, UT : 3,	CONFIG : 'F U T, 0, 0, 0',
	X =  -103.816  mm,	Y =   296.692  mm,	Z =     0.000  mm,
	W =  -167.361 deg,	P =     0.004 deg,	R =  -145.598 deg
};
P[2236]{
   GP1:
	UF : 7, UT : 3,	CONFIG : 'F U T, 0, 0, 0',
	X =  -103.816  mm,	Y =   296.692  mm,	Z =     0.000  mm,
	W =  -167.361 deg,	P =     0.004 deg,	R =  -145.598 deg
};
P[2237]{
   GP1:
	UF : 7, UT : 3,	CONFIG : 'F U T, 0, 0, 0',
	X =  -103.816  mm,	Y =   296.692  mm,	Z =     0.000  mm,
	W =  -167.361 deg,	P =     0.004 deg,	R =  -145.598 deg
};
P[2238]{
   GP1:
	UF : 7, UT : 3,	CONFIG : 'F U T, 0, 0, 0',
	X =  -103.816  mm,	Y =   296.692  mm,	Z =     0.000  mm,
	W =  -167.361 deg,	P =     0.004 deg,	R =  -145.598 deg
};
P[2239]{
   GP1:
	UF : 7, UT : 3,	CONFIG : 'F U T, 0, 0, 0',
	X =  -167.232  mm,	Y =   266.148  mm,	Z =     0.000  mm,
	W =  -167.365 deg,	P =    -0.022 deg,	R =  -132.938 deg
};
P[2240]{
   GP1:
	UF : 7, UT : 3,	CONFIG : 'F U T, 0, 0, 0',
	X =  -167.232  mm,	Y =   266.148  mm,	Z =     0.000  mm,
	W =  -167.365 deg,	P =    -0.022 deg,	R =  -132.938 deg
};
P[2241]{
   GP1:
	UF : 7, UT : 3,	CONFIG : 'F U T, 0, 0, 0',
	X =  -167.232  mm,	Y =   266.148  mm,	Z =     0.000  mm,
	W =  -167.365 deg,	P =    -0.022 deg,	R =  -132.938 deg
};
P[2242]{
   GP1:
	UF : 7, UT : 3,	CONFIG : 'F U T, 0, 0, 0',
	X =  -167.232  mm,	Y =   266.148  mm,	Z =     0.000  mm,
	W =  -167.365 deg,	P =    -0.022 deg,	R =  -132.938 deg
};
P[2243]{
   GP1:
	UF : 7, UT : 3,	CONFIG : 'F U T, 0, 0, 0',
	X =  -183.114  mm,	Y =   255.488  mm,	Z =     0.011  mm,
	W =  -167.354 deg,	P =    -0.024 deg,	R =  -129.291 deg
};
P[2244]{
   GP1:
	UF : 7, UT : 3,	CONFIG : 'F U T, 0, 0, 0',
	X =  -198.763  mm,	Y =   243.515  mm,	Z =     0.023  mm,
	W =  -167.343 deg,	P =    -0.029 deg,	R =  -125.737 deg
};
P[2245]{
   GP1:
	UF : 7, UT : 3,	CONFIG : 'F U T, 0, 0, 0',
	X =  -211.069  mm,	Y =   232.923  mm,	Z =     0.022  mm,
	W =  -167.329 deg,	P =     0.048 deg,	R =  -122.698 deg
};
P[2246]{
   GP1:
	UF : 7, UT : 3,	CONFIG : 'F U T, 0, 0, 0',
	X =  -222.261  mm,	Y =   222.261  mm,	Z =     0.000  mm,
	W =  -167.307 deg,	P =     0.119 deg,	R =  -119.437 deg
};
P[2247]{
   GP1:
	UF : 7, UT : 3,	CONFIG : 'F U T, 0, 0, 0',
	X =  -222.261  mm,	Y =   222.261  mm,	Z =     0.000  mm,
	W =  -167.307 deg,	P =     0.119 deg,	R =  -119.437 deg
};
P[2248]{
   GP1:
	UF : 7, UT : 3,	CONFIG : 'F U T, 0, 0, 0',
	X =  -222.261  mm,	Y =   222.261  mm,	Z =     0.000  mm,
	W =  -167.307 deg,	P =     0.119 deg,	R =  -119.437 deg
};
P[2249]{
   GP1:
	UF : 7, UT : 3,	CONFIG : 'F U T, 0, 0, 0',
	X =  -222.261  mm,	Y =   222.261  mm,	Z =     0.000  mm,
	W =  -167.307 deg,	P =     0.119 deg,	R =  -119.437 deg
};
P[2250]{
   GP1:
	UF : 7, UT : 3,	CONFIG : 'F U T, 0, 0, 0',
	X =  -266.148  mm,	Y =   167.232  mm,	Z =     0.000  mm,
	W =  -167.451 deg,	P =    -1.057 deg,	R =  -107.603 deg
};
P[2251]{
   GP1:
	UF : 7, UT : 3,	CONFIG : 'F U T, 0, 0, 0',
	X =  -266.148  mm,	Y =   167.232  mm,	Z =     0.000  mm,
	W =  -167.451 deg,	P =    -1.057 deg,	R =  -107.603 deg
};
P[2252]{
   GP1:
	UF : 7, UT : 3,	CONFIG : 'F U T, 0, 0, 0',
	X =  -266.148  mm,	Y =   167.232  mm,	Z =     0.000  mm,
	W =  -167.451 deg,	P =    -1.057 deg,	R =  -107.603 deg
};
P[2253]{
   GP1:
	UF : 7, UT : 3,	CONFIG : 'F U T, 0, 0, 0',
	X =  -266.148  mm,	Y =   167.232  mm,	Z =     0.000  mm,
	W =  -167.451 deg,	P =    -1.057 deg,	R =  -107.603 deg
};
P[2254]{
   GP1:
	UF : 7, UT : 3,	CONFIG : 'F U T, 0, 0, 0',
	X =  -269.323  mm,	Y =   162.065  mm,	Z =     0.117  mm,
	W =  -167.681 deg,	P =    -1.097 deg,	R =  -105.987 deg
};
P[2255]{
   GP1:
	UF : 7, UT : 3,	CONFIG : 'F U T, 0, 0, 0',
	X =  -277.022  mm,	Y =   148.536  mm,	Z =     0.388  mm,
	W =  -168.155 deg,	P =    -0.523 deg,	R =  -103.206 deg
};
P[2256]{
   GP1:
	UF : 7, UT : 3,	CONFIG : 'F U T, 0, 0, 0',
	X =  -285.722  mm,	Y =   131.011  mm,	Z =     0.439  mm,
	W =  -168.148 deg,	P =     0.621 deg,	R =   -99.624 deg
};
P[2257]{
   GP1:
	UF : 7, UT : 3,	CONFIG : 'F U T, 0, 0, 0',
	X =  -290.703  mm,	Y =   119.560  mm,	Z =     0.270  mm,
	W =  -167.700 deg,	P =     1.177 deg,	R =   -97.280 deg
};
P[2258]{
   GP1:
	UF : 7, UT : 3,	CONFIG : 'F U T, 0, 0, 0',
	X =  -292.713  mm,	Y =   114.575  mm,	Z =     0.169  mm,
	W =  -167.445 deg,	P =     1.139 deg,	R =   -96.303 deg
};
P[2259]{
   GP1:
	UF : 7, UT : 3,	CONFIG : 'F U T, 0, 0, 0',
	X =  -296.692  mm,	Y =   103.818  mm,	Z =     0.000  mm,
	W =  -167.160 deg,	P =     0.453 deg,	R =   -94.516 deg
};
P[2260]{
   GP1:
	UF : 7, UT : 3,	CONFIG : 'F U T, 0, 0, 0',
	X =  -296.692  mm,	Y =   103.818  mm,	Z =     0.000  mm,
	W =  -167.160 deg,	P =     0.453 deg,	R =   -94.516 deg
};
P[2261]{
   GP1:
	UF : 7, UT : 3,	CONFIG : 'F U T, 0, 0, 0',
	X =  -296.692  mm,	Y =   103.818  mm,	Z =     0.000  mm,
	W =  -167.160 deg,	P =     0.453 deg,	R =   -94.516 deg
};
P[2262]{
   GP1:
	UF : 7, UT : 3,	CONFIG : 'F U T, 0, 0, 0',
	X =  -296.692  mm,	Y =   103.818  mm,	Z =     0.000  mm,
	W =  -167.160 deg,	P =     0.453 deg,	R =   -94.516 deg
};
P[2263]{
   GP1:
	UF : 7, UT : 3,	CONFIG : 'F U T, 0, 1, 0',
	X =  -312.363  mm,	Y =    35.193  mm,	Z =     0.000  mm,
	W =  -167.364 deg,	P =    -0.010 deg,	R =   -80.974 deg
};
P[2264]{
   GP1:
	UF : 7, UT : 3,	CONFIG : 'F U T, 0, 1, 0',
	X =  -312.363  mm,	Y =    35.193  mm,	Z =     0.000  mm,
	W =  -167.364 deg,	P =    -0.010 deg,	R =   -80.974 deg
};
P[2265]{
   GP1:
	UF : 7, UT : 3,	CONFIG : 'F U T, 0, 1, 0',
	X =  -312.363  mm,	Y =    35.193  mm,	Z =     0.000  mm,
	W =  -167.364 deg,	P =    -0.010 deg,	R =   -80.974 deg
};
P[2266]{
   GP1:
	UF : 7, UT : 3,	CONFIG : 'F U T, 0, 1, 0',
	X =  -312.363  mm,	Y =    35.193  mm,	Z =     0.000  mm,
	W =  -167.364 deg,	P =    -0.010 deg,	R =   -80.974 deg
};
P[2267]{
   GP1:
	UF : 7, UT : 3,	CONFIG : 'F U T, 0, 1, 0',
	X =  -313.784  mm,	Y =    18.505  mm,	Z =     0.001  mm,
	W =  -167.364 deg,	P =    -0.002 deg,	R =   -78.279 deg
};
P[2268]{
   GP1:
	UF : 7, UT : 3,	CONFIG : 'F U T, 0, 1, 0',
	X =  -314.344  mm,	Y =     0.000  mm,	Z =     0.000  mm,
	W =  -167.362 deg,	P =     0.006 deg,	R =   -75.585 deg
};
P[2269]{
   GP1:
	UF : 7, UT : 3,	CONFIG : 'F U T, 0, 1, 0',
	X =  -314.344  mm,	Y =     0.000  mm,	Z =     0.000  mm,
	W =  -167.362 deg,	P =     0.006 deg,	R =   -75.585 deg
};
P[2270]{
   GP1:
	UF : 7, UT : 3,	CONFIG : 'F U T, 0, 1, 0',
	X =  -314.344  mm,	Y =     0.000  mm,	Z =     0.000  mm,
	W =  -167.362 deg,	P =     0.006 deg,	R =   -75.585 deg
};
P[2271]{
   GP1:
	UF : 7, UT : 3,	CONFIG : 'F U T, 0, 1, 0',
	X =  -314.344  mm,	Y =     0.000  mm,	Z =     0.000  mm,
	W =  -167.362 deg,	P =     0.006 deg,	R =   -75.585 deg
};
P[2272]{
   GP1:
	UF : 7, UT : 3,	CONFIG : 'F U T, 0, 1, 0',
	X =  -311.210  mm,	Y =     0.000  mm,	Z =     0.000  mm,
	W =  -167.362 deg,	P =     0.005 deg,	R =   -75.574 deg
};
P[2273]{
   GP1:
	UF : 7, UT : 3,	CONFIG : 'F U T, 0, 1, 0',
	X =  -311.210  mm,	Y =     0.000  mm,	Z =     0.000  mm,
	W =  -167.362 deg,	P =     0.005 deg,	R =   -75.574 deg
};
P[2274]{
   GP1:
	UF : 7, UT : 3,	CONFIG : 'F U T, 0, 1, 0',
	X =  -311.210  mm,	Y =     0.000  mm,	Z =     0.000  mm,
	W =  -167.362 deg,	P =     0.005 deg,	R =   -75.574 deg
};
P[2275]{
   GP1:
	UF : 7, UT : 3,	CONFIG : 'F U T, 0, 1, 0',
	X =  -311.210  mm,	Y =     0.000  mm,	Z =     0.000  mm,
	W =  -167.362 deg,	P =     0.005 deg,	R =   -75.574 deg
};
P[2276]{
   GP1:
	UF : 7, UT : 3,	CONFIG : 'F U T, 0, 1, 0',
	X =  -310.609  mm,	Y =    19.167  mm,	Z =     0.001  mm,
	W =  -167.363 deg,	P =    -0.003 deg,	R =   -78.435 deg
};
P[2277]{
   GP1:
	UF : 7, UT : 3,	CONFIG : 'F U T, 0, 1, 0',
	X =  -309.165  mm,	Y =    35.521  mm,	Z =     0.000  mm,
	W =  -167.364 deg,	P =    -0.010 deg,	R =   -81.404 deg
};
P[2278]{
   GP1:
	UF : 7, UT : 3,	CONFIG : 'F U T, 0, 1, 0',
	X =  -309.165  mm,	Y =    35.521  mm,	Z =     0.000  mm,
	W =  -167.364 deg,	P =    -0.010 deg,	R =   -81.404 deg
};
P[2279]{
   GP1:
	UF : 7, UT : 3,	CONFIG : 'F U T, 0, 1, 0',
	X =  -309.165  mm,	Y =    35.521  mm,	Z =     0.000  mm,
	W =  -167.364 deg,	P =    -0.010 deg,	R =   -81.404 deg
};
P[2280]{
   GP1:
	UF : 7, UT : 3,	CONFIG : 'F U T, 0, 1, 0',
	X =  -309.165  mm,	Y =    35.521  mm,	Z =     0.000  mm,
	W =  -167.364 deg,	P =    -0.010 deg,	R =   -81.404 deg
};
P[2281]{
   GP1:
	UF : 7, UT : 3,	CONFIG : 'F U T, 0, 0, 0',
	X =  -293.963  mm,	Y =   102.140  mm,	Z =     0.000  mm,
	W =  -167.168 deg,	P =     0.349 deg,	R =   -94.592 deg
};
P[2282]{
   GP1:
	UF : 7, UT : 3,	CONFIG : 'F U T, 0, 0, 0',
	X =  -293.963  mm,	Y =   102.140  mm,	Z =     0.000  mm,
	W =  -167.168 deg,	P =     0.349 deg,	R =   -94.592 deg
};
P[2283]{
   GP1:
	UF : 7, UT : 3,	CONFIG : 'F U T, 0, 0, 0',
	X =  -293.963  mm,	Y =   102.140  mm,	Z =     0.000  mm,
	W =  -167.168 deg,	P =     0.349 deg,	R =   -94.592 deg
};
P[2284]{
   GP1:
	UF : 7, UT : 3,	CONFIG : 'F U T, 0, 0, 0',
	X =  -293.963  mm,	Y =   102.140  mm,	Z =     0.000  mm,
	W =  -167.168 deg,	P =     0.349 deg,	R =   -94.592 deg
};
P[2285]{
   GP1:
	UF : 7, UT : 3,	CONFIG : 'F U T, 0, 0, 0',
	X =  -289.713  mm,	Y =   113.629  mm,	Z =     0.153  mm,
	W =  -167.448 deg,	P =     0.997 deg,	R =   -96.337 deg
};
P[2286]{
   GP1:
	UF : 7, UT : 3,	CONFIG : 'F U T, 0, 0, 0',
	X =  -285.444  mm,	Y =   123.944  mm,	Z =     0.328  mm,
	W =  -167.908 deg,	P =     0.905 deg,	R =   -98.395 deg
};
P[2287]{
   GP1:
	UF : 7, UT : 3,	CONFIG : 'F U T, 0, 0, 0',
	X =  -278.233  mm,	Y =   139.399  mm,	Z =     0.413  mm,
	W =  -168.175 deg,	P =     0.054 deg,	R =  -101.560 deg
};
P[2288]{
   GP1:
	UF : 7, UT : 3,	CONFIG : 'F U T, 0, 0, 0',
	X =  -270.057  mm,	Y =   154.632  mm,	Z =     0.235  mm,
	W =  -167.853 deg,	P =    -0.831 deg,	R =  -104.757 deg
};
P[2289]{
   GP1:
	UF : 7, UT : 3,	CONFIG : 'F U T, 0, 0, 0',
	X =  -263.128  mm,	Y =   166.143  mm,	Z =     0.000  mm,
	W =  -167.353 deg,	P =    -0.982 deg,	R =  -107.921 deg
};
P[2290]{
   GP1:
	UF : 7, UT : 3,	CONFIG : 'F U T, 0, 0, 0',
	X =  -263.128  mm,	Y =   166.143  mm,	Z =     0.000  mm,
	W =  -167.353 deg,	P =    -0.982 deg,	R =  -107.921 deg
};
P[2291]{
   GP1:
	UF : 7, UT : 3,	CONFIG : 'F U T, 0, 0, 0',
	X =  -263.128  mm,	Y =   166.143  mm,	Z =     0.000  mm,
	W =  -167.353 deg,	P =    -0.982 deg,	R =  -107.921 deg
};
P[2292]{
   GP1:
	UF : 7, UT : 3,	CONFIG : 'F U T, 0, 0, 0',
	X =  -263.128  mm,	Y =   166.143  mm,	Z =     0.000  mm,
	W =  -167.353 deg,	P =    -0.982 deg,	R =  -107.921 deg
};
P[2293]{
   GP1:
	UF : 7, UT : 3,	CONFIG : 'F U T, 0, 0, 0',
	X =  -220.529  mm,	Y =   219.561  mm,	Z =     0.000  mm,
	W =  -167.294 deg,	P =     0.118 deg,	R =  -119.493 deg
};
P[2294]{
   GP1:
	UF : 7, UT : 3,	CONFIG : 'F U T, 0, 0, 0',
	X =  -220.529  mm,	Y =   219.561  mm,	Z =     0.000  mm,
	W =  -167.294 deg,	P =     0.118 deg,	R =  -119.493 deg
};
P[2295]{
   GP1:
	UF : 7, UT : 3,	CONFIG : 'F U T, 0, 0, 0',
	X =  -220.529  mm,	Y =   219.561  mm,	Z =     0.000  mm,
	W =  -167.294 deg,	P =     0.118 deg,	R =  -119.493 deg
};
P[2296]{
   GP1:
	UF : 7, UT : 3,	CONFIG : 'F U T, 0, 0, 0',
	X =  -220.529  mm,	Y =   219.561  mm,	Z =     0.000  mm,
	W =  -167.294 deg,	P =     0.118 deg,	R =  -119.493 deg
};
P[2297]{
   GP1:
	UF : 7, UT : 3,	CONFIG : 'F U T, 0, 0, 0',
	X =  -208.972  mm,	Y =   230.595  mm,	Z =     0.023  mm,
	W =  -167.322 deg,	P =     0.047 deg,	R =  -122.742 deg
};
P[2298]{
   GP1:
	UF : 7, UT : 3,	CONFIG : 'F U T, 0, 0, 0',
	X =  -196.378  mm,	Y =   241.419  mm,	Z =     0.024  mm,
	W =  -167.342 deg,	P =    -0.031 deg,	R =  -125.847 deg
};
P[2299]{
   GP1:
	UF : 7, UT : 3,	CONFIG : 'F U T, 0, 0, 0',
	X =  -181.152  mm,	Y =   253.038  mm,	Z =     0.012  mm,
	W =  -167.352 deg,	P =    -0.027 deg,	R =  -129.328 deg
};
P[2300]{
   GP1:
	UF : 7, UT : 3,	CONFIG : 'F U T, 0, 0, 0',
	X =  -164.987  mm,	Y =   263.859  mm,	Z =     0.000  mm,
	W =  -167.364 deg,	P =    -0.024 deg,	R =  -132.775 deg
};
P[2301]{
   GP1:
	UF : 7, UT : 3,	CONFIG : 'F U T, 0, 0, 0',
	X =  -164.987  mm,	Y =   263.859  mm,	Z =     0.000  mm,
	W =  -167.364 deg,	P =    -0.024 deg,	R =  -132.775 deg
};
P[2302]{
   GP1:
	UF : 7, UT : 3,	CONFIG : 'F U T, 0, 0, 0',
	X =  -164.987  mm,	Y =   263.859  mm,	Z =     0.000  mm,
	W =  -167.364 deg,	P =    -0.024 deg,	R =  -132.775 deg
};
P[2303]{
   GP1:
	UF : 7, UT : 3,	CONFIG : 'F U T, 0, 0, 0',
	X =  -164.987  mm,	Y =   263.859  mm,	Z =     0.000  mm,
	W =  -167.364 deg,	P =    -0.024 deg,	R =  -132.775 deg
};
P[2304]{
   GP1:
	UF : 7, UT : 3,	CONFIG : 'F U T, 0, 0, 0',
	X =  -103.426  mm,	Y =   293.504  mm,	Z =     0.000  mm,
	W =  -167.361 deg,	P =     0.005 deg,	R =  -145.207 deg
};
P[2305]{
   GP1:
	UF : 7, UT : 3,	CONFIG : 'F U T, 0, 0, 0',
	X =  -103.426  mm,	Y =   293.504  mm,	Z =     0.000  mm,
	W =  -167.361 deg,	P =     0.005 deg,	R =  -145.207 deg
};
P[2306]{
   GP1:
	UF : 7, UT : 3,	CONFIG : 'F U T, 0, 0, 0',
	X =  -103.426  mm,	Y =   293.504  mm,	Z =     0.000  mm,
	W =  -167.361 deg,	P =     0.005 deg,	R =  -145.207 deg
};
P[2307]{
   GP1:
	UF : 7, UT : 3,	CONFIG : 'F U T, 0, 0, 0',
	X =  -103.426  mm,	Y =   293.504  mm,	Z =     0.000  mm,
	W =  -167.361 deg,	P =     0.005 deg,	R =  -145.207 deg
};
P[2308]{
   GP1:
	UF : 7, UT : 3,	CONFIG : 'F U T, 0, 0, 0',
	X =   -87.653  mm,	Y =   298.599  mm,	Z =     0.001  mm,
	W =  -167.362 deg,	P =     0.003 deg,	R =  -148.621 deg
};
P[2309]{
   GP1:
	UF : 7, UT : 3,	CONFIG : 'F U T, 0, 0, 0',
	X =   -70.707  mm,	Y =   303.056  mm,	Z =     0.001  mm,
	W =  -167.362 deg,	P =     0.002 deg,	R =  -151.841 deg
};
P[2310]{
   GP1:
	UF : 7, UT : 3,	CONFIG : 'F U T, 0, 0, 0',
	X =   -53.533  mm,	Y =   306.560  mm,	Z =     0.001  mm,
	W =  -167.363 deg,	P =     0.000 deg,	R =  -155.049 deg
};
P[2311]{
   GP1:
	UF : 7, UT : 3,	CONFIG : 'F U T, 0, 0, 0',
	X =   -34.169  mm,	Y =   309.326  mm,	Z =     0.000  mm,
	W =  -167.363 deg,	P =    -0.002 deg,	R =  -158.094 deg
};
P[2312]{
   GP1:
	UF : 7, UT : 3,	CONFIG : 'F U T, 0, 0, 0',
	X =   -34.169  mm,	Y =   309.326  mm,	Z =     0.000  mm,
	W =  -167.363 deg,	P =    -0.002 deg,	R =  -158.094 deg
};
P[2313]{
   GP1:
	UF : 7, UT : 3,	CONFIG : 'F U T, 0, 0, 0',
	X =   -34.169  mm,	Y =   309.326  mm,	Z =     0.000  mm,
	W =  -167.363 deg,	P =    -0.002 deg,	R =  -158.094 deg
};
P[2314]{
   GP1:
	UF : 7, UT : 3,	CONFIG : 'F U T, 0, 0, 0',
	X =   -34.169  mm,	Y =   309.326  mm,	Z =     0.000  mm,
	W =  -167.363 deg,	P =    -0.002 deg,	R =  -158.094 deg
};
P[2315]{
   GP1:
	UF : 7, UT : 3,	CONFIG : 'F U T, 0, 0, 0',
	X =    34.169  mm,	Y =   309.326  mm,	Z =     0.000  mm,
	W =  -167.363 deg,	P =     0.001 deg,	R =  -171.797 deg
};
P[2316]{
   GP1:
	UF : 7, UT : 3,	CONFIG : 'F U T, 0, 0, 0',
	X =    34.169  mm,	Y =   309.326  mm,	Z =     0.000  mm,
	W =  -167.363 deg,	P =     0.001 deg,	R =  -171.797 deg
};
P[2317]{
   GP1:
	UF : 7, UT : 3,	CONFIG : 'F U T, 0, 0, 0',
	X =    34.169  mm,	Y =   309.326  mm,	Z =     0.000  mm,
	W =  -167.363 deg,	P =     0.001 deg,	R =  -171.797 deg
};
P[2318]{
   GP1:
	UF : 7, UT : 3,	CONFIG : 'F U T, 0, 0, 0',
	X =    34.169  mm,	Y =   309.326  mm,	Z =     0.000  mm,
	W =  -167.363 deg,	P =     0.001 deg,	R =  -171.797 deg
};
P[2319]{
   GP1:
	UF : 7, UT : 3,	CONFIG : 'F U T, 0, 0, 0',
	X =    53.482  mm,	Y =   306.568  mm,	Z =     0.000  mm,
	W =  -167.363 deg,	P =     0.000 deg,	R =  -174.856 deg
};
P[2320]{
   GP1:
	UF : 7, UT : 3,	CONFIG : 'F U T, 0, 0, 0',
	X =    70.739  mm,	Y =   303.048  mm,	Z =     0.000  mm,
	W =  -167.363 deg,	P =     0.000 deg,	R =  -178.048 deg
};
P[2321]{
   GP1:
	UF : 7, UT : 3,	CONFIG : 'F U T, 0, 0, 0',
	X =    87.613  mm,	Y =   298.610  mm,	Z =     0.000  mm,
	W =  -167.363 deg,	P =    -0.001 deg,	R =   178.718 deg
};
P[2322]{
   GP1:
	UF : 7, UT : 3,	CONFIG : 'F U T, 0, 0, 0',
	X =   103.426  mm,	Y =   293.504  mm,	Z =     0.000  mm,
	W =  -167.363 deg,	P =    -0.001 deg,	R =   175.314 deg
};
P[2323]{
   GP1:
	UF : 7, UT : 3,	CONFIG : 'F U T, 0, 0, 0',
	X =   103.426  mm,	Y =   293.504  mm,	Z =     0.000  mm,
	W =  -167.363 deg,	P =    -0.001 deg,	R =   175.314 deg
};
P[2324]{
   GP1:
	UF : 7, UT : 3,	CONFIG : 'F U T, 0, 0, 0',
	X =   103.426  mm,	Y =   293.504  mm,	Z =     0.000  mm,
	W =  -167.363 deg,	P =    -0.001 deg,	R =   175.314 deg
};
P[2325]{
   GP1:
	UF : 7, UT : 3,	CONFIG : 'F U T, 0, 0, 0',
	X =   103.426  mm,	Y =   293.504  mm,	Z =     0.000  mm,
	W =  -167.363 deg,	P =    -0.001 deg,	R =   175.314 deg
};
P[2326]{
   GP1:
	UF : 7, UT : 3,	CONFIG : 'F U T, 0, 0, 0',
	X =   164.987  mm,	Y =   263.859  mm,	Z =     0.000  mm,
	W =  -167.362 deg,	P =     0.002 deg,	R =   162.852 deg
};
P[2327]{
   GP1:
	UF : 7, UT : 3,	CONFIG : 'F U T, 0, 0, 0',
	X =   164.987  mm,	Y =   263.859  mm,	Z =     0.000  mm,
	W =  -167.362 deg,	P =     0.002 deg,	R =   162.852 deg
};
P[2328]{
   GP1:
	UF : 7, UT : 3,	CONFIG : 'F U T, 0, 0, 0',
	X =   164.987  mm,	Y =   263.859  mm,	Z =     0.000  mm,
	W =  -167.362 deg,	P =     0.002 deg,	R =   162.852 deg
};
P[2329]{
   GP1:
	UF : 7, UT : 3,	CONFIG : 'F U T, 0, 0, 0',
	X =   164.987  mm,	Y =   263.859  mm,	Z =     0.000  mm,
	W =  -167.362 deg,	P =     0.002 deg,	R =   162.852 deg
};
P[2330]{
   GP1:
